// TIA Portal V16 export
// export: Created 2024-05-10T06:46:41.5011859Z, ExportSetting WithDefaults, DisplayName Totally Integrated Automation Portal, DisplayVersion V16, DisplayName TIA Portal Version Control Interface, DisplayVersion V16, DisplayName TIA Portal Openness, DisplayVersion V16, DisplayName STEP 7 Professional, DisplayVersion V16, DisplayName STEP 7 Safety, DisplayVersion V16, DisplayName WinCC Professional, DisplayVersion V16
FUNCTION_BLOCK "K04_报警"   // FB4, LAD
{ S7_Optimized_Access := 'TRUE' }
VERSION : 0.1
// stored: AutoNumber false, IsIECCheckEnabled false, IsRetainMemResEnabled false, MemoryReserve 100, SetENOAutomatically false, UDAEnableTagReadback false
   VAR
      MT_ErrTime : Array[1..3] of IEC_TIMER;   // 故障延迟
   END_VAR
   VAR_TEMP
      "W_All EMO" : Int;   // 急停报警汇总
      "W_All SLC" : Int;   // 光栅报警汇总
      "W_All DSW" : Int;   // 门保报警汇总
      "W_All OtherSafe" : Int;   // 其它安全报警汇总
      "W_All AirALM" : Int;   // 气压报警汇总
      "W_All DrumALM" : Array[1..3] of Int;   // 滚筒故障汇总
      "W_All DrumTiOver" : Array[1..3] of Int;   // 滚筒超时汇总
      "W_All InvALM" : Int;   // 变频器故障汇总
      "W_All InvNoRun" : Int;   // 变频器未运行故障汇总
      "W_All InvOverload" : Int;   // 变频器过载故障汇总
      "W_All InvTiOver" : Int;   // 变频器超时故障汇总
      "W_All ValAdvTiOver" : Array[1..3] of Int;   // 阀出动作超时汇总
      "W_All ValRetTiOver" : Array[1..3] of Int;   // 阀回动作超时汇总
      "W_All ValSensALM" : Array[1..3] of Int;   // 阀到位传感器都ON故障汇总
      "W_All ValSenCroALM" : Array[1..3] of Int;   // 阀到位传感器交叉ON故障汇总
      "W_All AxisALM" : Int;   // 轴报警汇总
      "W_All AxisERR" : Int;   // 轴故障汇总
      "W_All AxisReady" : Int;   // 轴未准备好汇总
      "W_All AxisHomeALM" : Int;   // 轴未回零故障汇总
      "W_All AxisNoRun" : Int;   // 轴未运行汇总
      "W_ALL AxisFLSALM" : Int;   // 轴正极限故障汇总
      "W_All AxisRLSALM" : Int;   // 轴负极限故障汇总
      "W_All RobotALM" : Int;   // 机器人故障汇总
      "W_All CCDALM" : Int;   // 视觉故障汇总
      "W_All CommALM" : Int;   // 通信故障汇总
      "W_All AnalogUpALM" : Int;   // 模拟量上限故障汇总
      "W_All AnalogLowALM" : Int;   // 模拟量下限故障汇总
      "W_All OtherALM" : Int;   // 其它故障汇总
      "W_All SensALM" : Array[1..6] of Int;   // 传感器故障汇总
      "W_All MoveALM" : Array[1..3] of Int;   // 动作异常汇总
      WD_RealTimeALM : Array[1..15] of DInt;   // 故障数据实时
      WD_OldTimeALM : Array[1..10] of DInt;   // 旧的故障
      WD_NewTimeALM : Array[1..10] of DInt;   // 新的故障
      M_SafeType : Bool;   // 安全类别
      M_AirType : Bool;   // 气压类别
      M_DrumType : Bool;   // 滚筒类别
      M_InvType : Bool;   // 变频器类类别
      M_ValType : Bool;   // 电磁阀类别
      M_ServoType : Bool;   // 伺服类别
      M_RoboType : Bool;   // 机器人类别
      M_CCDType : Bool;   // 视觉类别
      M_CommType : Bool;   // 通信类别
      M_AnalogType : Bool;   // 模拟量类别
      M_OtherType : Bool;   // 其它类别
      M_SensType : Bool;   // 传感器类
      M_MoveType : Bool;   // 动作异常类
      "M_All ALM" : Bool;   // 故障汇总
      "M_All NewALM" : Bool;   // 故障汇总新的
      M_BuzzeClose : Bool;   // 故障BZ关闭
      M_Pluse : Array[1..3] of Bool;   // 脉冲
   END_VAR
   VAR_TEMP   // added for the SCL form of the ladder/FBD networks
      _w1 : Bool;
      _w2 : Bool;
      _w3 : Bool;
      _w4 : Bool;
      _w5 : Bool;
      _w6 : Bool;
      _w7 : Bool;
      _w8 : Bool;
      _w9 : Bool;
      _w10 : Bool;
      _w11 : Bool;
      _w12 : Bool;
      _w13 : Bool;
      _w14 : Bool;
      _w15 : Bool;
      _w16 : Bool;
      _w17 : Bool;
      _w18 : Bool;
      _w19 : Bool;
      _w20 : Bool;
      _w21 : Bool;
      _w22 : Bool;
      _w23 : Bool;
      _w24 : Bool;
      _w25 : Bool;
      _w26 : Bool;
      _w27 : Bool;
      _w28 : Bool;
      _w29 : Bool;
      _w30 : Bool;
      _w31 : Bool;
      _w32 : Bool;
      _w33 : Bool;
      _w34 : Bool;
   END_VAR
BEGIN

REGION Network 1: 急停报警16个
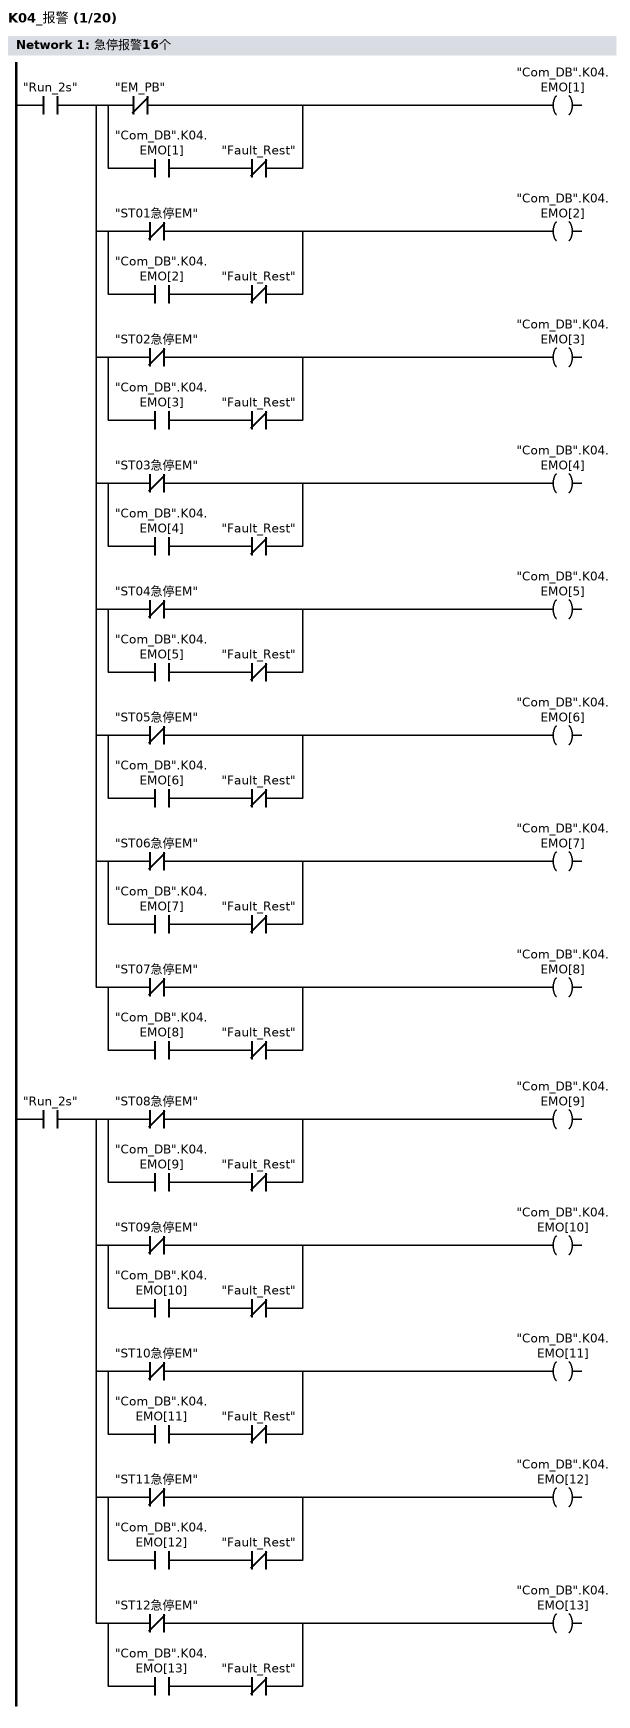
   RUNG wire#powerrail
      Contact( "Run_2s" )
      wire#w1
      I_Contact( "EM_PB" )
      wire#w2
      Coil( "Com_DB".K04.EMO[1] )
   END_RUNG
   RUNG wire#w1
      Contact( "Com_DB".K04.EMO[1] )
      I_Contact( "Fault_Rest" )
   END_RUNG wire#w2
   RUNG wire#w1
      I_Contact( "ST01急停EM" )
      wire#w3
      Coil( "Com_DB".K04.EMO[2] )
   END_RUNG
   RUNG wire#w1
      Contact( "Com_DB".K04.EMO[2] )
      I_Contact( "Fault_Rest" )
   END_RUNG wire#w3
   RUNG wire#w1
      I_Contact( "ST02急停EM" )
      wire#w4
      Coil( "Com_DB".K04.EMO[3] )
   END_RUNG
   RUNG wire#w1
      Contact( "Com_DB".K04.EMO[3] )
      I_Contact( "Fault_Rest" )
   END_RUNG wire#w4
   RUNG wire#w1
      I_Contact( "ST03急停EM" )
      wire#w5
      Coil( "Com_DB".K04.EMO[4] )
   END_RUNG
   RUNG wire#w1
      Contact( "Com_DB".K04.EMO[4] )
      I_Contact( "Fault_Rest" )
   END_RUNG wire#w5
   RUNG wire#w1
      I_Contact( "ST04急停EM" )
      wire#w6
      Coil( "Com_DB".K04.EMO[5] )
   END_RUNG
   RUNG wire#w1
      Contact( "Com_DB".K04.EMO[5] )
      I_Contact( "Fault_Rest" )
   END_RUNG wire#w6
   RUNG wire#w1
      I_Contact( "ST05急停EM" )
      wire#w7
      Coil( "Com_DB".K04.EMO[6] )
   END_RUNG
   RUNG wire#w1
      Contact( "Com_DB".K04.EMO[6] )
      I_Contact( "Fault_Rest" )
   END_RUNG wire#w7
   RUNG wire#w1
      I_Contact( "ST06急停EM" )
      wire#w8
      Coil( "Com_DB".K04.EMO[7] )
   END_RUNG
   RUNG wire#w1
      Contact( "Com_DB".K04.EMO[7] )
      I_Contact( "Fault_Rest" )
   END_RUNG wire#w8
   RUNG wire#w1
      I_Contact( "ST07急停EM" )
      wire#w9
      Coil( "Com_DB".K04.EMO[8] )
   END_RUNG
   RUNG wire#w1
      Contact( "Com_DB".K04.EMO[8] )
      I_Contact( "Fault_Rest" )
   END_RUNG wire#w9
   RUNG wire#powerrail
      Contact( "Run_2s" )
      wire#w10
      I_Contact( "ST08急停EM" )
      wire#w11
      Coil( "Com_DB".K04.EMO[9] )
   END_RUNG
   RUNG wire#w10
      Contact( "Com_DB".K04.EMO[9] )
      I_Contact( "Fault_Rest" )
   END_RUNG wire#w11
   RUNG wire#w10
      I_Contact( "ST09急停EM" )
      wire#w12
      Coil( "Com_DB".K04.EMO[10] )
   END_RUNG
   RUNG wire#w10
      Contact( "Com_DB".K04.EMO[10] )
      I_Contact( "Fault_Rest" )
   END_RUNG wire#w12
   RUNG wire#w10
      I_Contact( "ST10急停EM" )
      wire#w13
      Coil( "Com_DB".K04.EMO[11] )
   END_RUNG
   RUNG wire#w10
      Contact( "Com_DB".K04.EMO[11] )
      I_Contact( "Fault_Rest" )
   END_RUNG wire#w13
   RUNG wire#w10
      I_Contact( "ST11急停EM" )
      wire#w14
      Coil( "Com_DB".K04.EMO[12] )
   END_RUNG
   RUNG wire#w10
      Contact( "Com_DB".K04.EMO[12] )
      I_Contact( "Fault_Rest" )
   END_RUNG wire#w14
   RUNG wire#w10
      I_Contact( "ST12急停EM" )
      wire#w15
      Coil( "Com_DB".K04.EMO[13] )
   END_RUNG
   RUNG wire#w10
      Contact( "Com_DB".K04.EMO[13] )
      I_Contact( "Fault_Rest" )
   END_RUNG wire#w15
   // the same network as SCL:
   "Com_DB".K04.EMO[1] := "Run_2s" AND (NOT "EM_PB" OR ("Com_DB".K04.EMO[1] AND NOT "Fault_Rest"));
   "Com_DB".K04.EMO[2] := "Run_2s" AND (NOT "ST01急停EM" OR ("Com_DB".K04.EMO[2] AND NOT "Fault_Rest"));
   "Com_DB".K04.EMO[3] := "Run_2s" AND (NOT "ST02急停EM" OR ("Com_DB".K04.EMO[3] AND NOT "Fault_Rest"));
   "Com_DB".K04.EMO[4] := "Run_2s" AND (NOT "ST03急停EM" OR ("Com_DB".K04.EMO[4] AND NOT "Fault_Rest"));
   "Com_DB".K04.EMO[5] := "Run_2s" AND (NOT "ST04急停EM" OR ("Com_DB".K04.EMO[5] AND NOT "Fault_Rest"));
   "Com_DB".K04.EMO[6] := "Run_2s" AND (NOT "ST05急停EM" OR ("Com_DB".K04.EMO[6] AND NOT "Fault_Rest"));
   "Com_DB".K04.EMO[7] := "Run_2s" AND (NOT "ST06急停EM" OR ("Com_DB".K04.EMO[7] AND NOT "Fault_Rest"));
   "Com_DB".K04.EMO[8] := "Run_2s" AND (NOT "ST07急停EM" OR ("Com_DB".K04.EMO[8] AND NOT "Fault_Rest"));
   "Com_DB".K04.EMO[9] := "Run_2s" AND (NOT "ST08急停EM" OR ("Com_DB".K04.EMO[9] AND NOT "Fault_Rest"));
   "Com_DB".K04.EMO[10] := "Run_2s" AND (NOT "ST09急停EM" OR ("Com_DB".K04.EMO[10] AND NOT "Fault_Rest"));
   "Com_DB".K04.EMO[11] := "Run_2s" AND (NOT "ST10急停EM" OR ("Com_DB".K04.EMO[11] AND NOT "Fault_Rest"));
   "Com_DB".K04.EMO[12] := "Run_2s" AND (NOT "ST11急停EM" OR ("Com_DB".K04.EMO[12] AND NOT "Fault_Rest"));
   "Com_DB".K04.EMO[13] := "Run_2s" AND (NOT "ST12急停EM" OR ("Com_DB".K04.EMO[13] AND NOT "Fault_Rest"));
END_REGION

REGION Network 2: 光栅报警16个
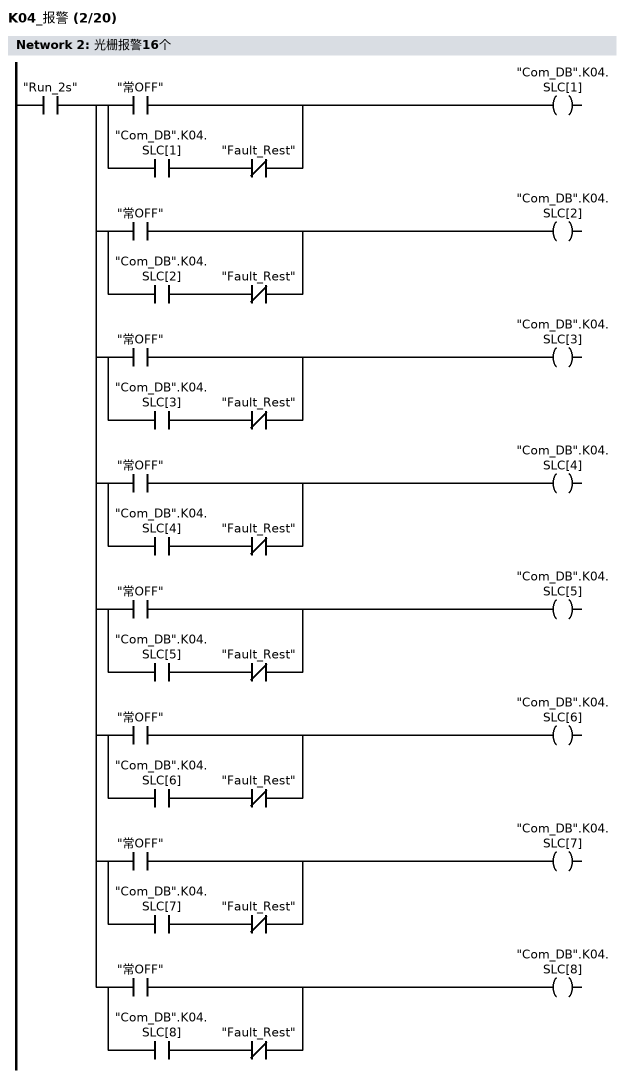
   RUNG wire#powerrail
      Contact( "Run_2s" )
      wire#w1
      Contact( "常OFF" )
      wire#w2
      Coil( "Com_DB".K04.SLC[1] )
   END_RUNG
   RUNG wire#w1
      Contact( "Com_DB".K04.SLC[1] )
      I_Contact( "Fault_Rest" )
   END_RUNG wire#w2
   RUNG wire#w1
      Contact( "常OFF" )
      wire#w3
      Coil( "Com_DB".K04.SLC[2] )
   END_RUNG
   RUNG wire#w1
      Contact( "Com_DB".K04.SLC[2] )
      I_Contact( "Fault_Rest" )
   END_RUNG wire#w3
   RUNG wire#w1
      Contact( "常OFF" )
      wire#w4
      Coil( "Com_DB".K04.SLC[3] )
   END_RUNG
   RUNG wire#w1
      Contact( "Com_DB".K04.SLC[3] )
      I_Contact( "Fault_Rest" )
   END_RUNG wire#w4
   RUNG wire#w1
      Contact( "常OFF" )
      wire#w5
      Coil( "Com_DB".K04.SLC[4] )
   END_RUNG
   RUNG wire#w1
      Contact( "Com_DB".K04.SLC[4] )
      I_Contact( "Fault_Rest" )
   END_RUNG wire#w5
   RUNG wire#w1
      Contact( "常OFF" )
      wire#w6
      Coil( "Com_DB".K04.SLC[5] )
   END_RUNG
   RUNG wire#w1
      Contact( "Com_DB".K04.SLC[5] )
      I_Contact( "Fault_Rest" )
   END_RUNG wire#w6
   RUNG wire#w1
      Contact( "常OFF" )
      wire#w7
      Coil( "Com_DB".K04.SLC[6] )
   END_RUNG
   RUNG wire#w1
      Contact( "Com_DB".K04.SLC[6] )
      I_Contact( "Fault_Rest" )
   END_RUNG wire#w7
   RUNG wire#w1
      Contact( "常OFF" )
      wire#w8
      Coil( "Com_DB".K04.SLC[7] )
   END_RUNG
   RUNG wire#w1
      Contact( "Com_DB".K04.SLC[7] )
      I_Contact( "Fault_Rest" )
   END_RUNG wire#w8
   RUNG wire#w1
      Contact( "常OFF" )
      wire#w9
      Coil( "Com_DB".K04.SLC[8] )
   END_RUNG
   RUNG wire#w1
      Contact( "Com_DB".K04.SLC[8] )
      I_Contact( "Fault_Rest" )
   END_RUNG wire#w9
   // the same network as SCL:
   "Com_DB".K04.SLC[1] := "Run_2s" AND ("常OFF" OR ("Com_DB".K04.SLC[1] AND NOT "Fault_Rest"));
   "Com_DB".K04.SLC[2] := "Run_2s" AND ("常OFF" OR ("Com_DB".K04.SLC[2] AND NOT "Fault_Rest"));
   "Com_DB".K04.SLC[3] := "Run_2s" AND ("常OFF" OR ("Com_DB".K04.SLC[3] AND NOT "Fault_Rest"));
   "Com_DB".K04.SLC[4] := "Run_2s" AND ("常OFF" OR ("Com_DB".K04.SLC[4] AND NOT "Fault_Rest"));
   "Com_DB".K04.SLC[5] := "Run_2s" AND ("常OFF" OR ("Com_DB".K04.SLC[5] AND NOT "Fault_Rest"));
   "Com_DB".K04.SLC[6] := "Run_2s" AND ("常OFF" OR ("Com_DB".K04.SLC[6] AND NOT "Fault_Rest"));
   "Com_DB".K04.SLC[7] := "Run_2s" AND ("常OFF" OR ("Com_DB".K04.SLC[7] AND NOT "Fault_Rest"));
   "Com_DB".K04.SLC[8] := "Run_2s" AND ("常OFF" OR ("Com_DB".K04.SLC[8] AND NOT "Fault_Rest"));
END_REGION

REGION Network 3: 门开关报警16个
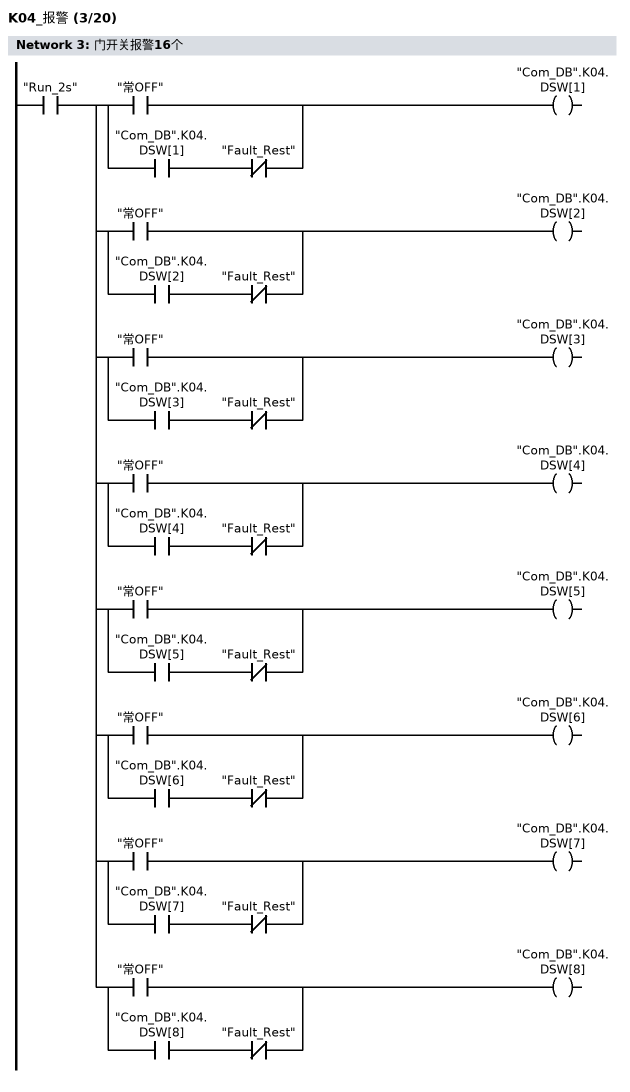
   RUNG wire#powerrail
      Contact( "Run_2s" )
      wire#w1
      Contact( "常OFF" )
      wire#w2
      Coil( "Com_DB".K04.DSW[1] )
   END_RUNG
   RUNG wire#w1
      Contact( "Com_DB".K04.DSW[1] )
      I_Contact( "Fault_Rest" )
   END_RUNG wire#w2
   RUNG wire#w1
      Contact( "常OFF" )
      wire#w3
      Coil( "Com_DB".K04.DSW[2] )
   END_RUNG
   RUNG wire#w1
      Contact( "Com_DB".K04.DSW[2] )
      I_Contact( "Fault_Rest" )
   END_RUNG wire#w3
   RUNG wire#w1
      Contact( "常OFF" )
      wire#w4
      Coil( "Com_DB".K04.DSW[3] )
   END_RUNG
   RUNG wire#w1
      Contact( "Com_DB".K04.DSW[3] )
      I_Contact( "Fault_Rest" )
   END_RUNG wire#w4
   RUNG wire#w1
      Contact( "常OFF" )
      wire#w5
      Coil( "Com_DB".K04.DSW[4] )
   END_RUNG
   RUNG wire#w1
      Contact( "Com_DB".K04.DSW[4] )
      I_Contact( "Fault_Rest" )
   END_RUNG wire#w5
   RUNG wire#w1
      Contact( "常OFF" )
      wire#w6
      Coil( "Com_DB".K04.DSW[5] )
   END_RUNG
   RUNG wire#w1
      Contact( "Com_DB".K04.DSW[5] )
      I_Contact( "Fault_Rest" )
   END_RUNG wire#w6
   RUNG wire#w1
      Contact( "常OFF" )
      wire#w7
      Coil( "Com_DB".K04.DSW[6] )
   END_RUNG
   RUNG wire#w1
      Contact( "Com_DB".K04.DSW[6] )
      I_Contact( "Fault_Rest" )
   END_RUNG wire#w7
   RUNG wire#w1
      Contact( "常OFF" )
      wire#w8
      Coil( "Com_DB".K04.DSW[7] )
   END_RUNG
   RUNG wire#w1
      Contact( "Com_DB".K04.DSW[7] )
      I_Contact( "Fault_Rest" )
   END_RUNG wire#w8
   RUNG wire#w1
      Contact( "常OFF" )
      wire#w9
      Coil( "Com_DB".K04.DSW[8] )
   END_RUNG
   RUNG wire#w1
      Contact( "Com_DB".K04.DSW[8] )
      I_Contact( "Fault_Rest" )
   END_RUNG wire#w9
   // the same network as SCL:
   "Com_DB".K04.DSW[1] := "Run_2s" AND ("常OFF" OR ("Com_DB".K04.DSW[1] AND NOT "Fault_Rest"));
   "Com_DB".K04.DSW[2] := "Run_2s" AND ("常OFF" OR ("Com_DB".K04.DSW[2] AND NOT "Fault_Rest"));
   "Com_DB".K04.DSW[3] := "Run_2s" AND ("常OFF" OR ("Com_DB".K04.DSW[3] AND NOT "Fault_Rest"));
   "Com_DB".K04.DSW[4] := "Run_2s" AND ("常OFF" OR ("Com_DB".K04.DSW[4] AND NOT "Fault_Rest"));
   "Com_DB".K04.DSW[5] := "Run_2s" AND ("常OFF" OR ("Com_DB".K04.DSW[5] AND NOT "Fault_Rest"));
   "Com_DB".K04.DSW[6] := "Run_2s" AND ("常OFF" OR ("Com_DB".K04.DSW[6] AND NOT "Fault_Rest"));
   "Com_DB".K04.DSW[7] := "Run_2s" AND ("常OFF" OR ("Com_DB".K04.DSW[7] AND NOT "Fault_Rest"));
   "Com_DB".K04.DSW[8] := "Run_2s" AND ("常OFF" OR ("Com_DB".K04.DSW[8] AND NOT "Fault_Rest"));
END_REGION

REGION Network 4: 其它安全报警16个Other types of security
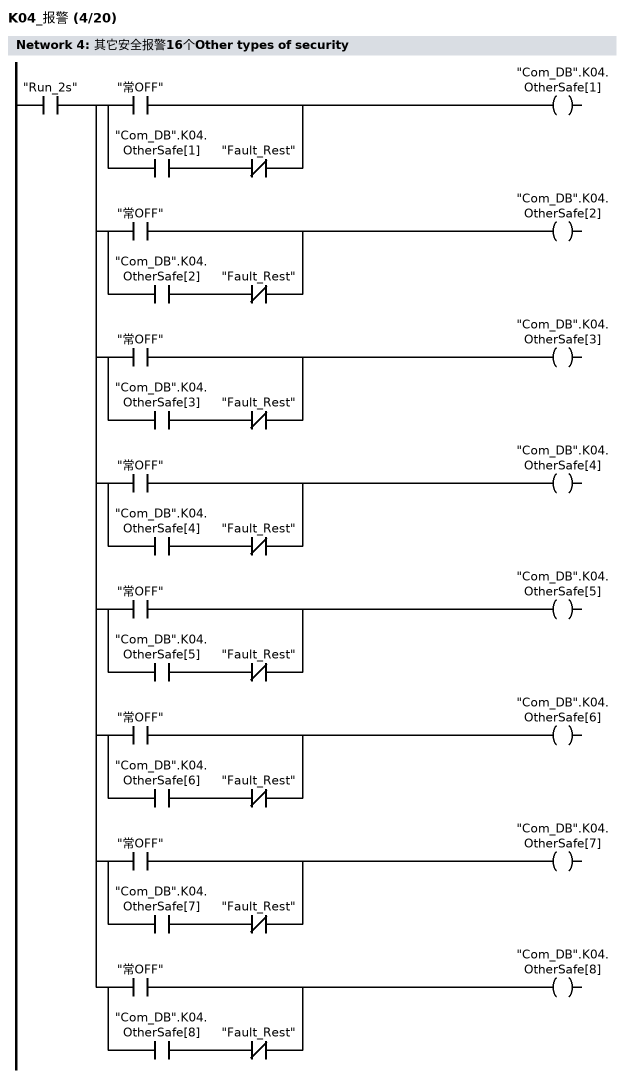
   RUNG wire#powerrail
      Contact( "Run_2s" )
      wire#w1
      Contact( "常OFF" )
      wire#w2
      Coil( "Com_DB".K04.OtherSafe[1] )
   END_RUNG
   RUNG wire#w1
      Contact( "Com_DB".K04.OtherSafe[1] )
      I_Contact( "Fault_Rest" )
   END_RUNG wire#w2
   RUNG wire#w1
      Contact( "常OFF" )
      wire#w3
      Coil( "Com_DB".K04.OtherSafe[2] )
   END_RUNG
   RUNG wire#w1
      Contact( "Com_DB".K04.OtherSafe[2] )
      I_Contact( "Fault_Rest" )
   END_RUNG wire#w3
   RUNG wire#w1
      Contact( "常OFF" )
      wire#w4
      Coil( "Com_DB".K04.OtherSafe[3] )
   END_RUNG
   RUNG wire#w1
      Contact( "Com_DB".K04.OtherSafe[3] )
      I_Contact( "Fault_Rest" )
   END_RUNG wire#w4
   RUNG wire#w1
      Contact( "常OFF" )
      wire#w5
      Coil( "Com_DB".K04.OtherSafe[4] )
   END_RUNG
   RUNG wire#w1
      Contact( "Com_DB".K04.OtherSafe[4] )
      I_Contact( "Fault_Rest" )
   END_RUNG wire#w5
   RUNG wire#w1
      Contact( "常OFF" )
      wire#w6
      Coil( "Com_DB".K04.OtherSafe[5] )
   END_RUNG
   RUNG wire#w1
      Contact( "Com_DB".K04.OtherSafe[5] )
      I_Contact( "Fault_Rest" )
   END_RUNG wire#w6
   RUNG wire#w1
      Contact( "常OFF" )
      wire#w7
      Coil( "Com_DB".K04.OtherSafe[6] )
   END_RUNG
   RUNG wire#w1
      Contact( "Com_DB".K04.OtherSafe[6] )
      I_Contact( "Fault_Rest" )
   END_RUNG wire#w7
   RUNG wire#w1
      Contact( "常OFF" )
      wire#w8
      Coil( "Com_DB".K04.OtherSafe[7] )
   END_RUNG
   RUNG wire#w1
      Contact( "Com_DB".K04.OtherSafe[7] )
      I_Contact( "Fault_Rest" )
   END_RUNG wire#w8
   RUNG wire#w1
      Contact( "常OFF" )
      wire#w9
      Coil( "Com_DB".K04.OtherSafe[8] )
   END_RUNG
   RUNG wire#w1
      Contact( "Com_DB".K04.OtherSafe[8] )
      I_Contact( "Fault_Rest" )
   END_RUNG wire#w9
   // the same network as SCL:
   "Com_DB".K04.OtherSafe[1] := "Run_2s" AND ("常OFF" OR ("Com_DB".K04.OtherSafe[1] AND NOT "Fault_Rest"));
   "Com_DB".K04.OtherSafe[2] := "Run_2s" AND ("常OFF" OR ("Com_DB".K04.OtherSafe[2] AND NOT "Fault_Rest"));
   "Com_DB".K04.OtherSafe[3] := "Run_2s" AND ("常OFF" OR ("Com_DB".K04.OtherSafe[3] AND NOT "Fault_Rest"));
   "Com_DB".K04.OtherSafe[4] := "Run_2s" AND ("常OFF" OR ("Com_DB".K04.OtherSafe[4] AND NOT "Fault_Rest"));
   "Com_DB".K04.OtherSafe[5] := "Run_2s" AND ("常OFF" OR ("Com_DB".K04.OtherSafe[5] AND NOT "Fault_Rest"));
   "Com_DB".K04.OtherSafe[6] := "Run_2s" AND ("常OFF" OR ("Com_DB".K04.OtherSafe[6] AND NOT "Fault_Rest"));
   "Com_DB".K04.OtherSafe[7] := "Run_2s" AND ("常OFF" OR ("Com_DB".K04.OtherSafe[7] AND NOT "Fault_Rest"));
   "Com_DB".K04.OtherSafe[8] := "Run_2s" AND ("常OFF" OR ("Com_DB".K04.OtherSafe[8] AND NOT "Fault_Rest"));
END_REGION

REGION Network 5: 气压低报警16个
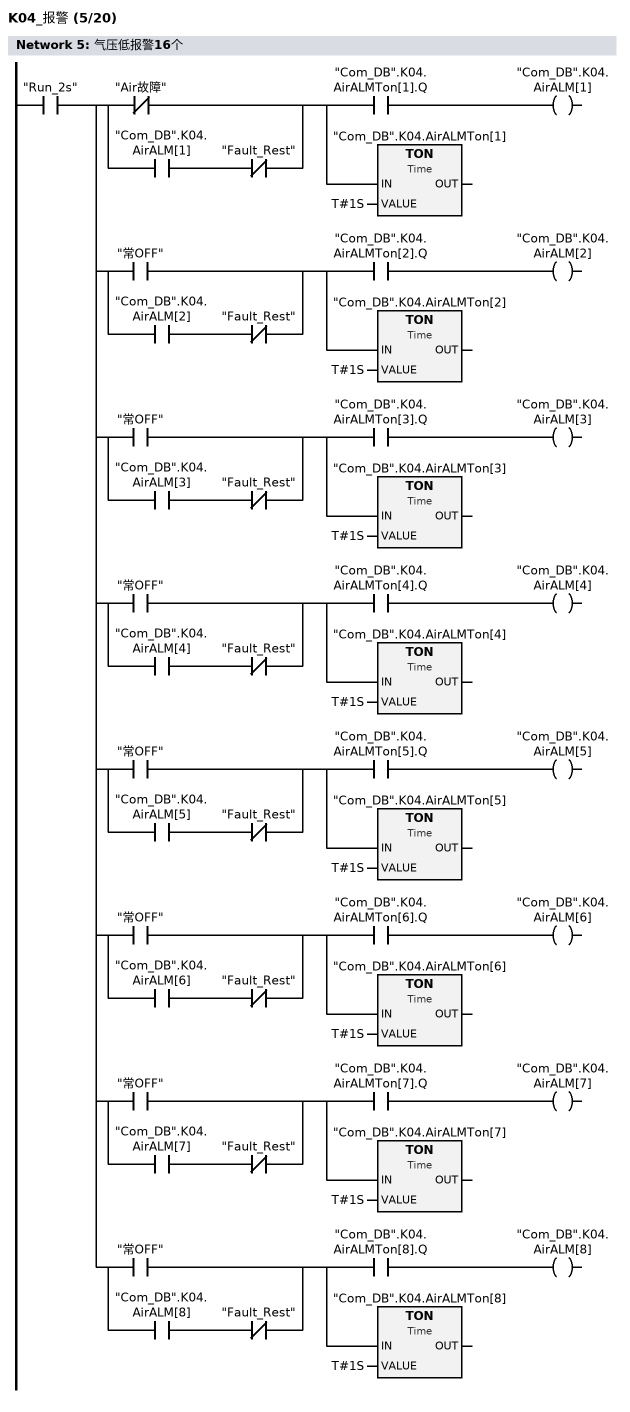
   #_w1 := "Run_2s" AND (NOT "Air故障" OR ("Com_DB".K04.AirALM[1] AND NOT "Fault_Rest"));
   "Com_DB".K04.AirALM[1] := #_w1 AND "Com_DB".K04.AirALMTon[1].Q;
   "Com_DB".K04.AirALMTon[1].TON(IN := #_w1, PT := T#1S);   // TON coil
   #_w2 := "Run_2s" AND ("常OFF" OR ("Com_DB".K04.AirALM[2] AND NOT "Fault_Rest"));
   "Com_DB".K04.AirALM[2] := #_w2 AND "Com_DB".K04.AirALMTon[2].Q;
   "Com_DB".K04.AirALMTon[2].TON(IN := #_w2, PT := T#1S);   // TON coil
   #_w3 := "Run_2s" AND ("常OFF" OR ("Com_DB".K04.AirALM[3] AND NOT "Fault_Rest"));
   "Com_DB".K04.AirALM[3] := #_w3 AND "Com_DB".K04.AirALMTon[3].Q;
   "Com_DB".K04.AirALMTon[3].TON(IN := #_w3, PT := T#1S);   // TON coil
   #_w4 := "Run_2s" AND ("常OFF" OR ("Com_DB".K04.AirALM[4] AND NOT "Fault_Rest"));
   "Com_DB".K04.AirALM[4] := #_w4 AND "Com_DB".K04.AirALMTon[4].Q;
   "Com_DB".K04.AirALMTon[4].TON(IN := #_w4, PT := T#1S);   // TON coil
   #_w5 := "Run_2s" AND ("常OFF" OR ("Com_DB".K04.AirALM[5] AND NOT "Fault_Rest"));
   "Com_DB".K04.AirALM[5] := #_w5 AND "Com_DB".K04.AirALMTon[5].Q;
   "Com_DB".K04.AirALMTon[5].TON(IN := #_w5, PT := T#1S);   // TON coil
   #_w6 := "Run_2s" AND ("常OFF" OR ("Com_DB".K04.AirALM[6] AND NOT "Fault_Rest"));
   "Com_DB".K04.AirALM[6] := #_w6 AND "Com_DB".K04.AirALMTon[6].Q;
   "Com_DB".K04.AirALMTon[6].TON(IN := #_w6, PT := T#1S);   // TON coil
   #_w7 := "Run_2s" AND ("常OFF" OR ("Com_DB".K04.AirALM[7] AND NOT "Fault_Rest"));
   "Com_DB".K04.AirALM[7] := #_w7 AND "Com_DB".K04.AirALMTon[7].Q;
   "Com_DB".K04.AirALMTon[7].TON(IN := #_w7, PT := T#1S);   // TON coil
   #_w8 := "Run_2s" AND ("常OFF" OR ("Com_DB".K04.AirALM[8] AND NOT "Fault_Rest"));
   "Com_DB".K04.AirALM[8] := #_w8 AND "Com_DB".K04.AirALMTon[8].Q;
   "Com_DB".K04.AirALMTon[8].TON(IN := #_w8, PT := T#1S);   // TON coil
END_REGION

REGION Network 6: 滚筒故障48个
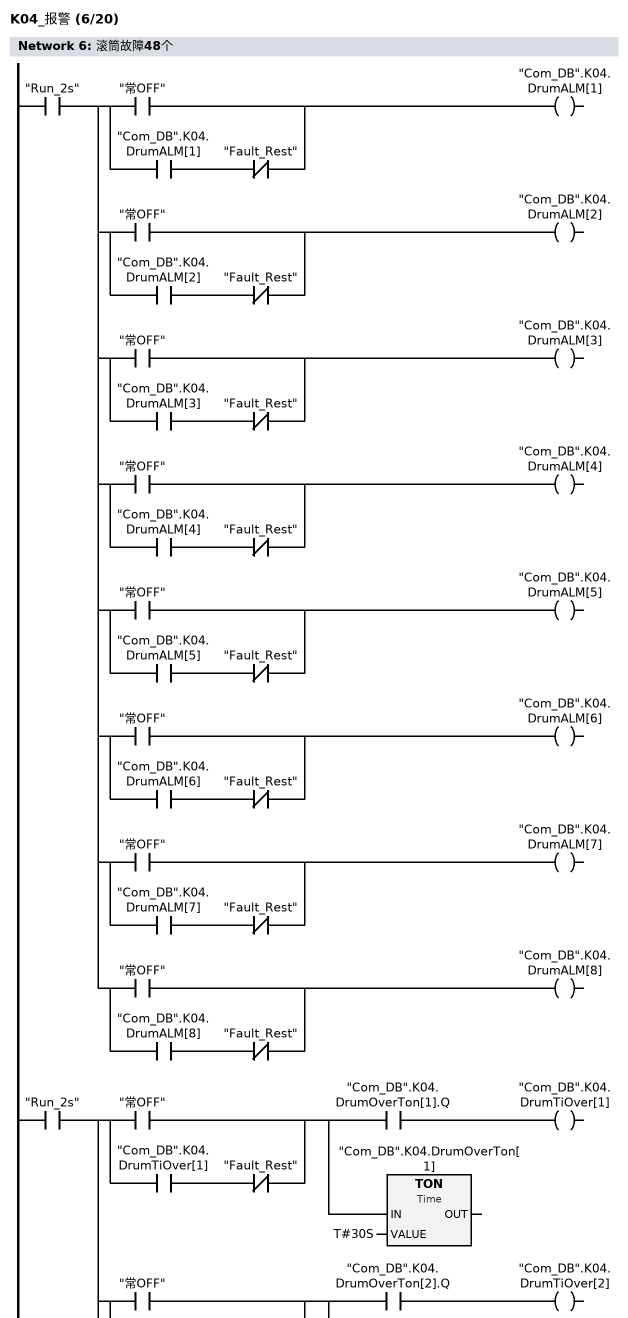
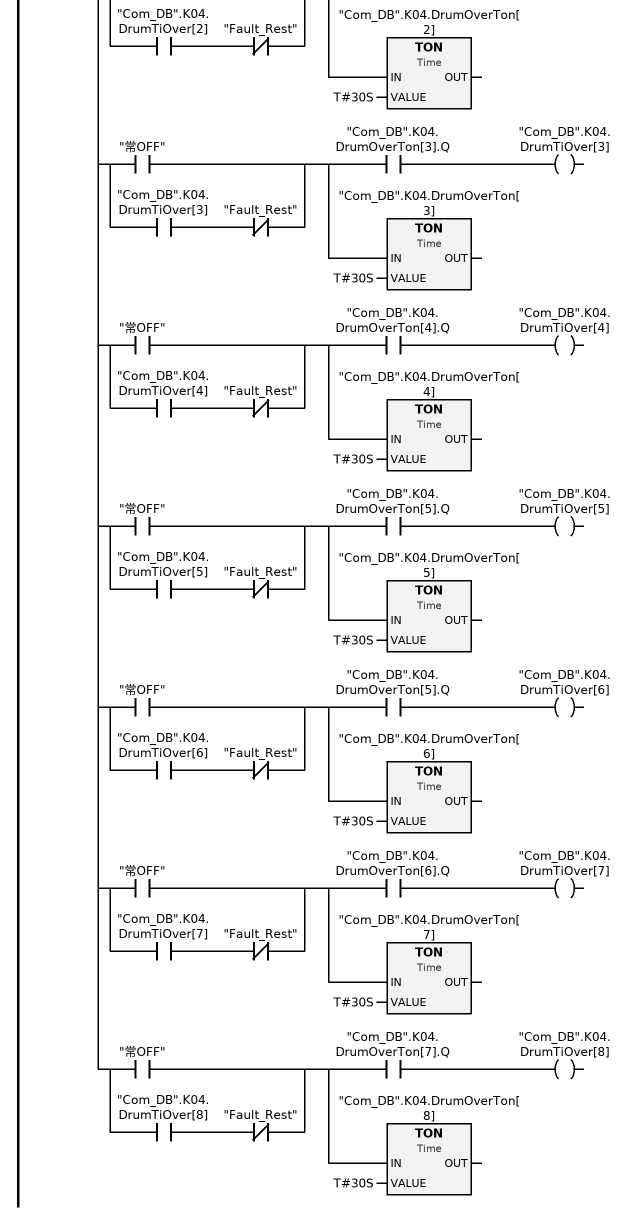
   "Com_DB".K04.DrumALM[1] := "Run_2s" AND ("常OFF" OR ("Com_DB".K04.DrumALM[1] AND NOT "Fault_Rest"));
   "Com_DB".K04.DrumALM[2] := "Run_2s" AND ("常OFF" OR ("Com_DB".K04.DrumALM[2] AND NOT "Fault_Rest"));
   "Com_DB".K04.DrumALM[3] := "Run_2s" AND ("常OFF" OR ("Com_DB".K04.DrumALM[3] AND NOT "Fault_Rest"));
   "Com_DB".K04.DrumALM[4] := "Run_2s" AND ("常OFF" OR ("Com_DB".K04.DrumALM[4] AND NOT "Fault_Rest"));
   "Com_DB".K04.DrumALM[5] := "Run_2s" AND ("常OFF" OR ("Com_DB".K04.DrumALM[5] AND NOT "Fault_Rest"));
   "Com_DB".K04.DrumALM[6] := "Run_2s" AND ("常OFF" OR ("Com_DB".K04.DrumALM[6] AND NOT "Fault_Rest"));
   "Com_DB".K04.DrumALM[7] := "Run_2s" AND ("常OFF" OR ("Com_DB".K04.DrumALM[7] AND NOT "Fault_Rest"));
   "Com_DB".K04.DrumALM[8] := "Run_2s" AND ("常OFF" OR ("Com_DB".K04.DrumALM[8] AND NOT "Fault_Rest"));
   #_w1 := "Run_2s" AND ("常OFF" OR ("Com_DB".K04.DrumTiOver[1] AND NOT "Fault_Rest"));
   "Com_DB".K04.DrumTiOver[1] := #_w1 AND "Com_DB".K04.DrumOverTon[1].Q;
   "Com_DB".K04.DrumOverTon[1].TON(IN := #_w1, PT := T#30S);   // TON coil
   #_w2 := "Run_2s" AND ("常OFF" OR ("Com_DB".K04.DrumTiOver[2] AND NOT "Fault_Rest"));
   "Com_DB".K04.DrumTiOver[2] := #_w2 AND "Com_DB".K04.DrumOverTon[2].Q;
   "Com_DB".K04.DrumOverTon[2].TON(IN := #_w2, PT := T#30S);   // TON coil
   #_w3 := "Run_2s" AND ("常OFF" OR ("Com_DB".K04.DrumTiOver[3] AND NOT "Fault_Rest"));
   "Com_DB".K04.DrumTiOver[3] := #_w3 AND "Com_DB".K04.DrumOverTon[3].Q;
   "Com_DB".K04.DrumOverTon[3].TON(IN := #_w3, PT := T#30S);   // TON coil
   #_w4 := "Run_2s" AND ("常OFF" OR ("Com_DB".K04.DrumTiOver[4] AND NOT "Fault_Rest"));
   "Com_DB".K04.DrumTiOver[4] := #_w4 AND "Com_DB".K04.DrumOverTon[4].Q;
   "Com_DB".K04.DrumOverTon[4].TON(IN := #_w4, PT := T#30S);   // TON coil
   #_w5 := "Run_2s" AND ("常OFF" OR ("Com_DB".K04.DrumTiOver[5] AND NOT "Fault_Rest"));
   "Com_DB".K04.DrumTiOver[5] := #_w5 AND "Com_DB".K04.DrumOverTon[5].Q;
   "Com_DB".K04.DrumOverTon[5].TON(IN := #_w5, PT := T#30S);   // TON coil
   #_w6 := "Run_2s" AND ("常OFF" OR ("Com_DB".K04.DrumTiOver[6] AND NOT "Fault_Rest"));
   "Com_DB".K04.DrumTiOver[6] := #_w6 AND "Com_DB".K04.DrumOverTon[5].Q;
   "Com_DB".K04.DrumOverTon[6].TON(IN := #_w6, PT := T#30S);   // TON coil
   #_w7 := "Run_2s" AND ("常OFF" OR ("Com_DB".K04.DrumTiOver[7] AND NOT "Fault_Rest"));
   "Com_DB".K04.DrumTiOver[7] := #_w7 AND "Com_DB".K04.DrumOverTon[6].Q;
   "Com_DB".K04.DrumOverTon[7].TON(IN := #_w7, PT := T#30S);   // TON coil
   #_w8 := "Run_2s" AND ("常OFF" OR ("Com_DB".K04.DrumTiOver[8] AND NOT "Fault_Rest"));
   "Com_DB".K04.DrumTiOver[8] := #_w8 AND "Com_DB".K04.DrumOverTon[7].Q;
   "Com_DB".K04.DrumOverTon[8].TON(IN := #_w8, PT := T#30S);   // TON coil
END_REGION

REGION Network 7: 变频器 异常/未运/超时/过载 16个
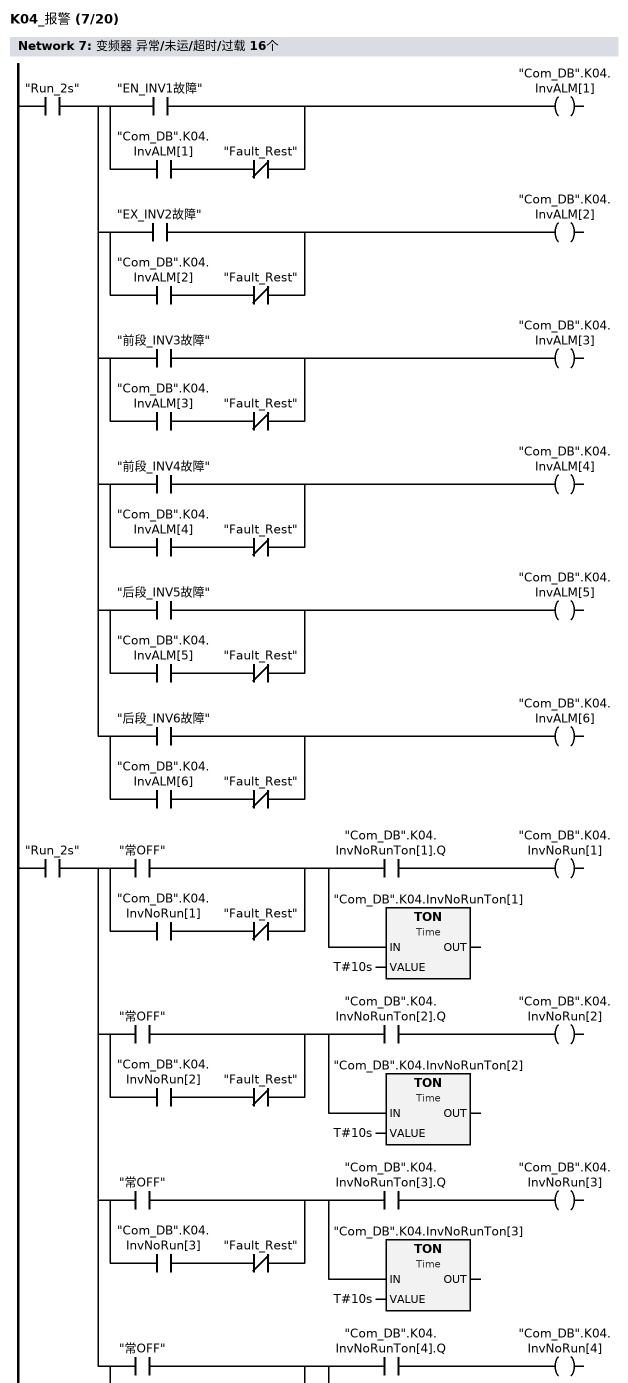
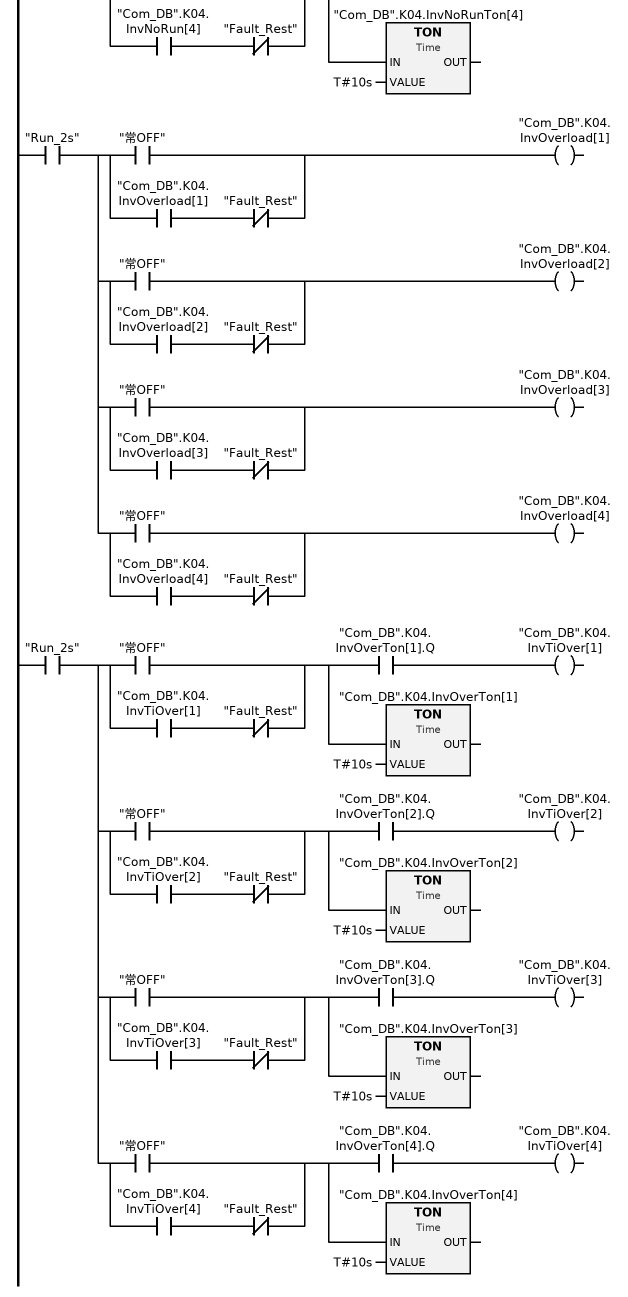
   "Com_DB".K04.InvALM[1] := "Run_2s" AND ("EN_INV1故障" OR ("Com_DB".K04.InvALM[1] AND NOT "Fault_Rest"));
   "Com_DB".K04.InvALM[2] := "Run_2s" AND ("EX_INV2故障" OR ("Com_DB".K04.InvALM[2] AND NOT "Fault_Rest"));
   "Com_DB".K04.InvALM[3] := "Run_2s" AND ("前段_INV3故障" OR ("Com_DB".K04.InvALM[3] AND NOT "Fault_Rest"));
   "Com_DB".K04.InvALM[4] := "Run_2s" AND ("前段_INV4故障" OR ("Com_DB".K04.InvALM[4] AND NOT "Fault_Rest"));
   "Com_DB".K04.InvALM[5] := "Run_2s" AND ("后段_INV5故障" OR ("Com_DB".K04.InvALM[5] AND NOT "Fault_Rest"));
   "Com_DB".K04.InvALM[6] := "Run_2s" AND ("后段_INV6故障" OR ("Com_DB".K04.InvALM[6] AND NOT "Fault_Rest"));
   #_w1 := "Run_2s" AND ("常OFF" OR ("Com_DB".K04.InvNoRun[1] AND NOT "Fault_Rest"));
   "Com_DB".K04.InvNoRun[1] := #_w1 AND "Com_DB".K04.InvNoRunTon[1].Q;
   "Com_DB".K04.InvNoRunTon[1].TON(IN := #_w1, PT := T#10s);   // TON coil
   #_w2 := "Run_2s" AND ("常OFF" OR ("Com_DB".K04.InvNoRun[2] AND NOT "Fault_Rest"));
   "Com_DB".K04.InvNoRun[2] := #_w2 AND "Com_DB".K04.InvNoRunTon[2].Q;
   "Com_DB".K04.InvNoRunTon[2].TON(IN := #_w2, PT := T#10s);   // TON coil
   #_w3 := "Run_2s" AND ("常OFF" OR ("Com_DB".K04.InvNoRun[3] AND NOT "Fault_Rest"));
   "Com_DB".K04.InvNoRun[3] := #_w3 AND "Com_DB".K04.InvNoRunTon[3].Q;
   "Com_DB".K04.InvNoRunTon[3].TON(IN := #_w3, PT := T#10s);   // TON coil
   #_w4 := "Run_2s" AND ("常OFF" OR ("Com_DB".K04.InvNoRun[4] AND NOT "Fault_Rest"));
   "Com_DB".K04.InvNoRun[4] := #_w4 AND "Com_DB".K04.InvNoRunTon[4].Q;
   "Com_DB".K04.InvNoRunTon[4].TON(IN := #_w4, PT := T#10s);   // TON coil
   "Com_DB".K04.InvOverload[1] := "Run_2s" AND ("常OFF" OR ("Com_DB".K04.InvOverload[1] AND NOT "Fault_Rest"));
   "Com_DB".K04.InvOverload[2] := "Run_2s" AND ("常OFF" OR ("Com_DB".K04.InvOverload[2] AND NOT "Fault_Rest"));
   "Com_DB".K04.InvOverload[3] := "Run_2s" AND ("常OFF" OR ("Com_DB".K04.InvOverload[3] AND NOT "Fault_Rest"));
   "Com_DB".K04.InvOverload[4] := "Run_2s" AND ("常OFF" OR ("Com_DB".K04.InvOverload[4] AND NOT "Fault_Rest"));
   #_w5 := "Run_2s" AND ("常OFF" OR ("Com_DB".K04.InvTiOver[1] AND NOT "Fault_Rest"));
   "Com_DB".K04.InvTiOver[1] := #_w5 AND "Com_DB".K04.InvOverTon[1].Q;
   "Com_DB".K04.InvOverTon[1].TON(IN := #_w5, PT := T#10s);   // TON coil
   #_w6 := "Run_2s" AND ("常OFF" OR ("Com_DB".K04.InvTiOver[2] AND NOT "Fault_Rest"));
   "Com_DB".K04.InvTiOver[2] := #_w6 AND "Com_DB".K04.InvOverTon[2].Q;
   "Com_DB".K04.InvOverTon[2].TON(IN := #_w6, PT := T#10s);   // TON coil
   #_w7 := "Run_2s" AND ("常OFF" OR ("Com_DB".K04.InvTiOver[3] AND NOT "Fault_Rest"));
   "Com_DB".K04.InvTiOver[3] := #_w7 AND "Com_DB".K04.InvOverTon[3].Q;
   "Com_DB".K04.InvOverTon[3].TON(IN := #_w7, PT := T#10s);   // TON coil
   #_w8 := "Run_2s" AND ("常OFF" OR ("Com_DB".K04.InvTiOver[4] AND NOT "Fault_Rest"));
   "Com_DB".K04.InvTiOver[4] := #_w8 AND "Com_DB".K04.InvOverTon[4].Q;
   "Com_DB".K04.InvOverTon[4].TON(IN := #_w8, PT := T#10s);   // TON coil
END_REGION

REGION Network 8: 气缸故障48个
   // 气缸故障FB库已经有输出故障，请在FB关联，这里不需写
END_REGION

REGION Network 9: 伺服故障16个伺服
   // 轴警告、轴错误FB库以及有输出，这里不需要写
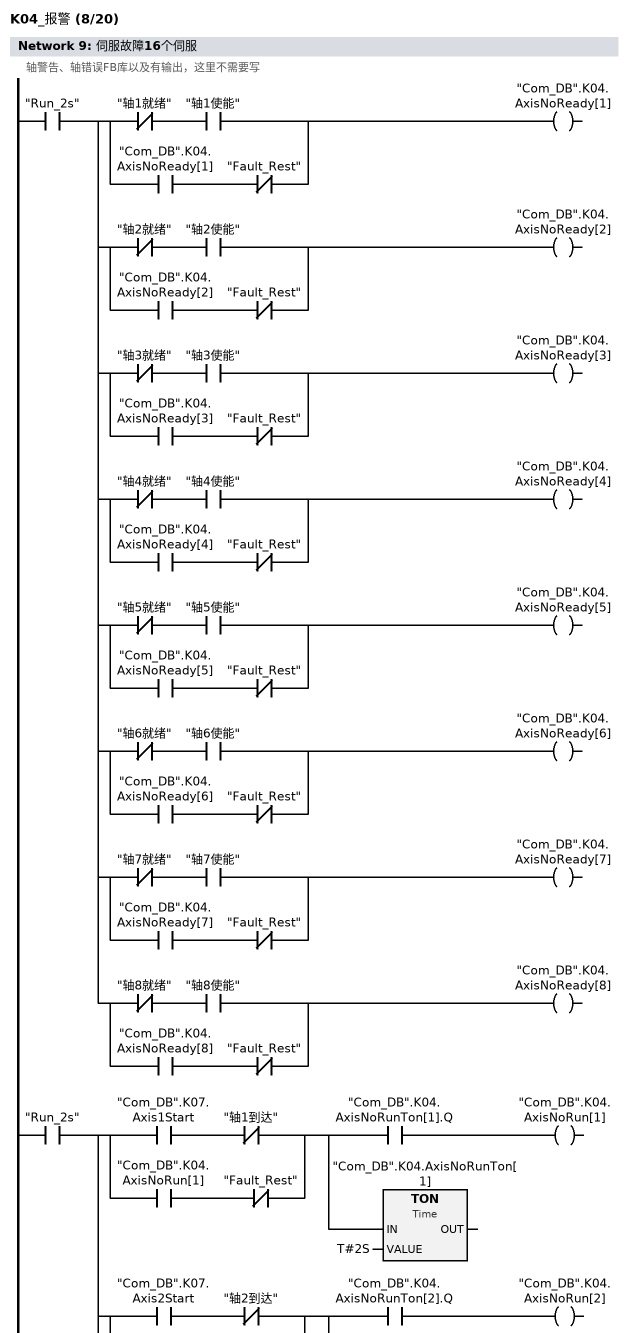
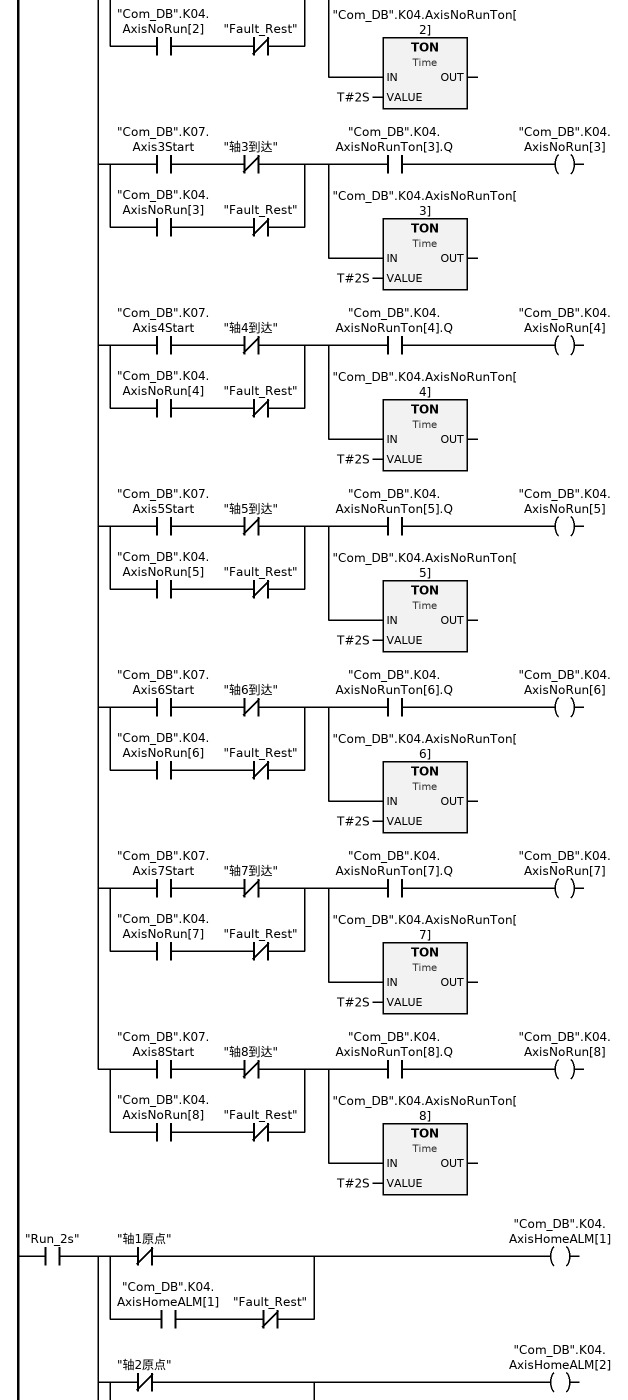
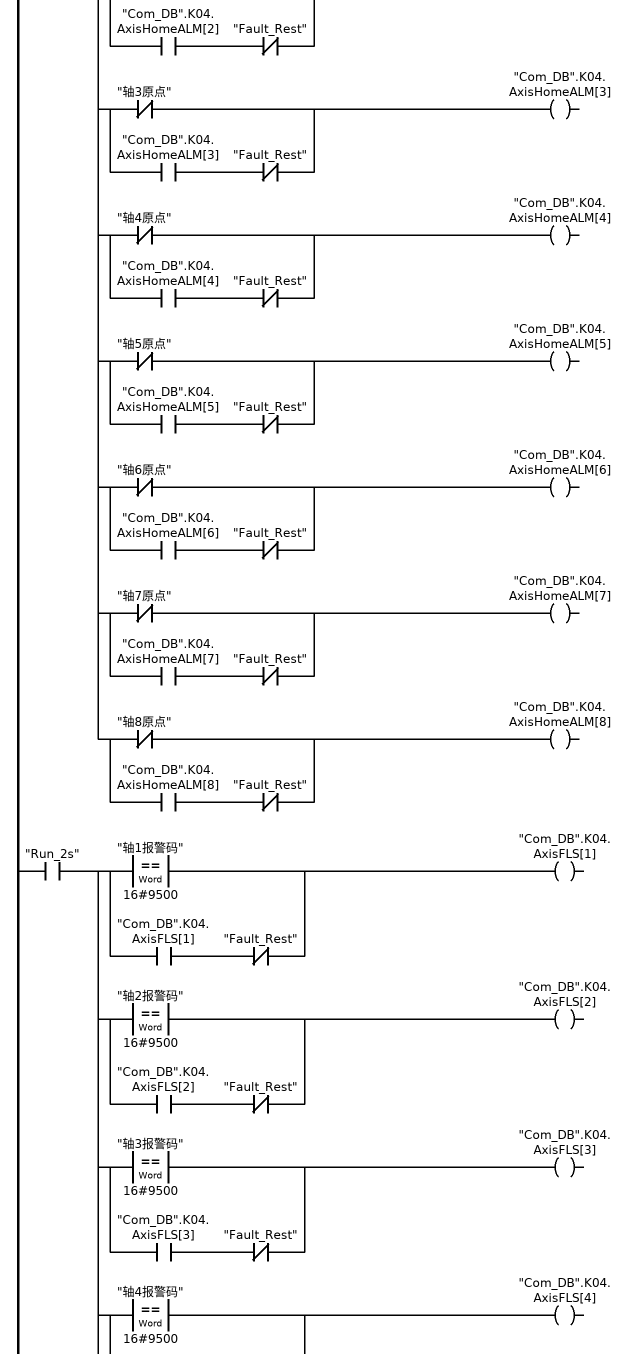
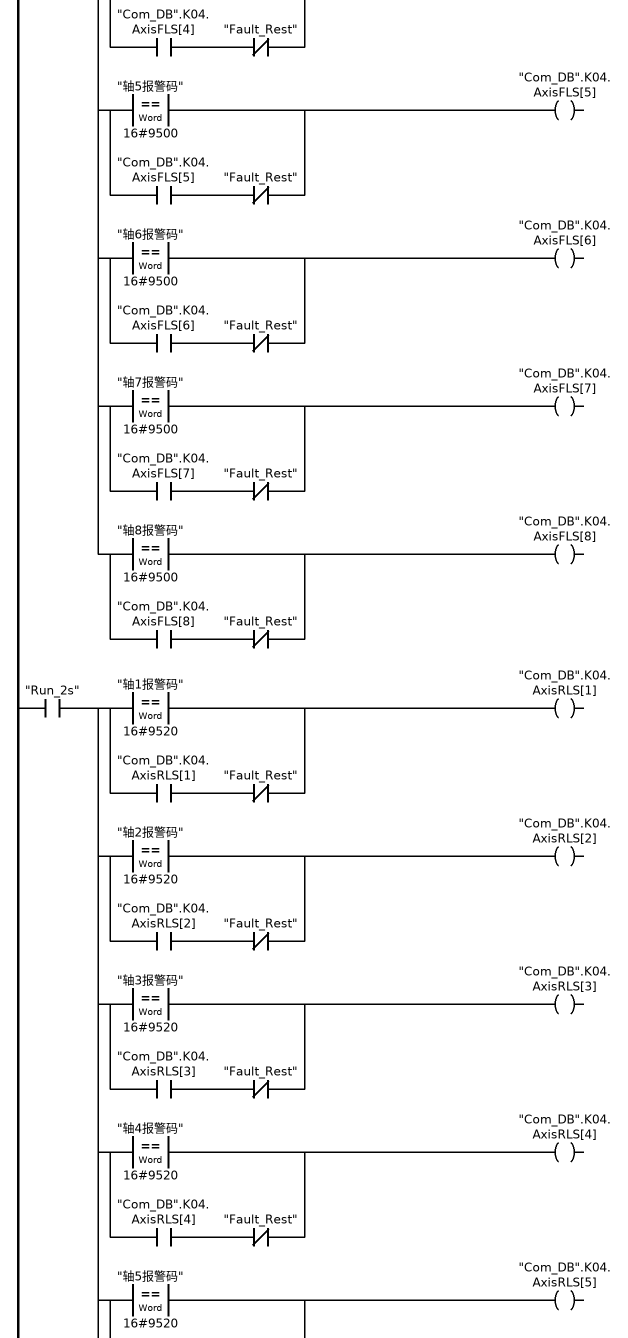
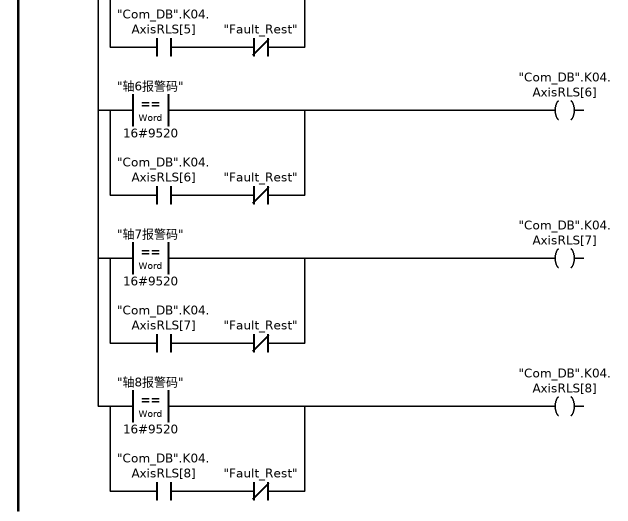
   "Com_DB".K04.AxisNoReady[1] := "Run_2s" AND ((NOT "轴1就绪" AND "轴1使能") OR ("Com_DB".K04.AxisNoReady[1] AND NOT "Fault_Rest"));
   "Com_DB".K04.AxisNoReady[2] := "Run_2s" AND ((NOT "轴2就绪" AND "轴2使能") OR ("Com_DB".K04.AxisNoReady[2] AND NOT "Fault_Rest"));
   "Com_DB".K04.AxisNoReady[3] := "Run_2s" AND ((NOT "轴3就绪" AND "轴3使能") OR ("Com_DB".K04.AxisNoReady[3] AND NOT "Fault_Rest"));
   "Com_DB".K04.AxisNoReady[4] := "Run_2s" AND ((NOT "轴4就绪" AND "轴4使能") OR ("Com_DB".K04.AxisNoReady[4] AND NOT "Fault_Rest"));
   "Com_DB".K04.AxisNoReady[5] := "Run_2s" AND ((NOT "轴5就绪" AND "轴5使能") OR ("Com_DB".K04.AxisNoReady[5] AND NOT "Fault_Rest"));
   "Com_DB".K04.AxisNoReady[6] := "Run_2s" AND ((NOT "轴6就绪" AND "轴6使能") OR ("Com_DB".K04.AxisNoReady[6] AND NOT "Fault_Rest"));
   "Com_DB".K04.AxisNoReady[7] := "Run_2s" AND ((NOT "轴7就绪" AND "轴7使能") OR ("Com_DB".K04.AxisNoReady[7] AND NOT "Fault_Rest"));
   "Com_DB".K04.AxisNoReady[8] := "Run_2s" AND ((NOT "轴8就绪" AND "轴8使能") OR ("Com_DB".K04.AxisNoReady[8] AND NOT "Fault_Rest"));
   #_w1 := "Run_2s" AND (("Com_DB".K07.Axis1Start AND NOT "轴1到达") OR ("Com_DB".K04.AxisNoRun[1] AND NOT "Fault_Rest"));
   "Com_DB".K04.AxisNoRun[1] := #_w1 AND "Com_DB".K04.AxisNoRunTon[1].Q;
   "Com_DB".K04.AxisNoRunTon[1].TON(IN := #_w1, PT := T#2S);   // TON coil
   #_w2 := "Run_2s" AND (("Com_DB".K07.Axis2Start AND NOT "轴2到达") OR ("Com_DB".K04.AxisNoRun[2] AND NOT "Fault_Rest"));
   "Com_DB".K04.AxisNoRun[2] := #_w2 AND "Com_DB".K04.AxisNoRunTon[2].Q;
   "Com_DB".K04.AxisNoRunTon[2].TON(IN := #_w2, PT := T#2S);   // TON coil
   #_w3 := "Run_2s" AND (("Com_DB".K07.Axis3Start AND NOT "轴3到达") OR ("Com_DB".K04.AxisNoRun[3] AND NOT "Fault_Rest"));
   "Com_DB".K04.AxisNoRun[3] := #_w3 AND "Com_DB".K04.AxisNoRunTon[3].Q;
   "Com_DB".K04.AxisNoRunTon[3].TON(IN := #_w3, PT := T#2S);   // TON coil
   #_w4 := "Run_2s" AND (("Com_DB".K07.Axis4Start AND NOT "轴4到达") OR ("Com_DB".K04.AxisNoRun[4] AND NOT "Fault_Rest"));
   "Com_DB".K04.AxisNoRun[4] := #_w4 AND "Com_DB".K04.AxisNoRunTon[4].Q;
   "Com_DB".K04.AxisNoRunTon[4].TON(IN := #_w4, PT := T#2S);   // TON coil
   #_w5 := "Run_2s" AND (("Com_DB".K07.Axis5Start AND NOT "轴5到达") OR ("Com_DB".K04.AxisNoRun[5] AND NOT "Fault_Rest"));
   "Com_DB".K04.AxisNoRun[5] := #_w5 AND "Com_DB".K04.AxisNoRunTon[5].Q;
   "Com_DB".K04.AxisNoRunTon[5].TON(IN := #_w5, PT := T#2S);   // TON coil
   #_w6 := "Run_2s" AND (("Com_DB".K07.Axis6Start AND NOT "轴6到达") OR ("Com_DB".K04.AxisNoRun[6] AND NOT "Fault_Rest"));
   "Com_DB".K04.AxisNoRun[6] := #_w6 AND "Com_DB".K04.AxisNoRunTon[6].Q;
   "Com_DB".K04.AxisNoRunTon[6].TON(IN := #_w6, PT := T#2S);   // TON coil
   #_w7 := "Run_2s" AND (("Com_DB".K07.Axis7Start AND NOT "轴7到达") OR ("Com_DB".K04.AxisNoRun[7] AND NOT "Fault_Rest"));
   "Com_DB".K04.AxisNoRun[7] := #_w7 AND "Com_DB".K04.AxisNoRunTon[7].Q;
   "Com_DB".K04.AxisNoRunTon[7].TON(IN := #_w7, PT := T#2S);   // TON coil
   #_w8 := "Run_2s" AND (("Com_DB".K07.Axis8Start AND NOT "轴8到达") OR ("Com_DB".K04.AxisNoRun[8] AND NOT "Fault_Rest"));
   "Com_DB".K04.AxisNoRun[8] := #_w8 AND "Com_DB".K04.AxisNoRunTon[8].Q;
   "Com_DB".K04.AxisNoRunTon[8].TON(IN := #_w8, PT := T#2S);   // TON coil
   "Com_DB".K04.AxisHomeALM[1] := "Run_2s" AND (NOT "轴1原点" OR ("Com_DB".K04.AxisHomeALM[1] AND NOT "Fault_Rest"));
   "Com_DB".K04.AxisHomeALM[2] := "Run_2s" AND (NOT "轴2原点" OR ("Com_DB".K04.AxisHomeALM[2] AND NOT "Fault_Rest"));
   "Com_DB".K04.AxisHomeALM[3] := "Run_2s" AND (NOT "轴3原点" OR ("Com_DB".K04.AxisHomeALM[3] AND NOT "Fault_Rest"));
   "Com_DB".K04.AxisHomeALM[4] := "Run_2s" AND (NOT "轴4原点" OR ("Com_DB".K04.AxisHomeALM[4] AND NOT "Fault_Rest"));
   "Com_DB".K04.AxisHomeALM[5] := "Run_2s" AND (NOT "轴5原点" OR ("Com_DB".K04.AxisHomeALM[5] AND NOT "Fault_Rest"));
   "Com_DB".K04.AxisHomeALM[6] := "Run_2s" AND (NOT "轴6原点" OR ("Com_DB".K04.AxisHomeALM[6] AND NOT "Fault_Rest"));
   "Com_DB".K04.AxisHomeALM[7] := "Run_2s" AND (NOT "轴7原点" OR ("Com_DB".K04.AxisHomeALM[7] AND NOT "Fault_Rest"));
   "Com_DB".K04.AxisHomeALM[8] := "Run_2s" AND (NOT "轴8原点" OR ("Com_DB".K04.AxisHomeALM[8] AND NOT "Fault_Rest"));
   "Com_DB".K04.AxisFLS[1] := "Run_2s" AND (("轴1报警码" = 16#9500) OR ("Com_DB".K04.AxisFLS[1] AND NOT "Fault_Rest"));
   "Com_DB".K04.AxisFLS[2] := "Run_2s" AND (("轴2报警码" = 16#9500) OR ("Com_DB".K04.AxisFLS[2] AND NOT "Fault_Rest"));
   "Com_DB".K04.AxisFLS[3] := "Run_2s" AND (("轴3报警码" = 16#9500) OR ("Com_DB".K04.AxisFLS[3] AND NOT "Fault_Rest"));
   "Com_DB".K04.AxisFLS[4] := "Run_2s" AND (("轴4报警码" = 16#9500) OR ("Com_DB".K04.AxisFLS[4] AND NOT "Fault_Rest"));
   "Com_DB".K04.AxisFLS[5] := "Run_2s" AND (("轴5报警码" = 16#9500) OR ("Com_DB".K04.AxisFLS[5] AND NOT "Fault_Rest"));
   "Com_DB".K04.AxisFLS[6] := "Run_2s" AND (("轴6报警码" = 16#9500) OR ("Com_DB".K04.AxisFLS[6] AND NOT "Fault_Rest"));
   "Com_DB".K04.AxisFLS[7] := "Run_2s" AND (("轴7报警码" = 16#9500) OR ("Com_DB".K04.AxisFLS[7] AND NOT "Fault_Rest"));
   "Com_DB".K04.AxisFLS[8] := "Run_2s" AND (("轴8报警码" = 16#9500) OR ("Com_DB".K04.AxisFLS[8] AND NOT "Fault_Rest"));
   "Com_DB".K04.AxisRLS[1] := "Run_2s" AND (("轴1报警码" = 16#9520) OR ("Com_DB".K04.AxisRLS[1] AND NOT "Fault_Rest"));
   "Com_DB".K04.AxisRLS[2] := "Run_2s" AND (("轴2报警码" = 16#9520) OR ("Com_DB".K04.AxisRLS[2] AND NOT "Fault_Rest"));
   "Com_DB".K04.AxisRLS[3] := "Run_2s" AND (("轴3报警码" = 16#9520) OR ("Com_DB".K04.AxisRLS[3] AND NOT "Fault_Rest"));
   "Com_DB".K04.AxisRLS[4] := "Run_2s" AND (("轴4报警码" = 16#9520) OR ("Com_DB".K04.AxisRLS[4] AND NOT "Fault_Rest"));
   "Com_DB".K04.AxisRLS[5] := "Run_2s" AND (("轴5报警码" = 16#9520) OR ("Com_DB".K04.AxisRLS[5] AND NOT "Fault_Rest"));
   "Com_DB".K04.AxisRLS[6] := "Run_2s" AND (("轴6报警码" = 16#9520) OR ("Com_DB".K04.AxisRLS[6] AND NOT "Fault_Rest"));
   "Com_DB".K04.AxisRLS[7] := "Run_2s" AND (("轴7报警码" = 16#9520) OR ("Com_DB".K04.AxisRLS[7] AND NOT "Fault_Rest"));
   "Com_DB".K04.AxisRLS[8] := "Run_2s" AND (("轴8报警码" = 16#9520) OR ("Com_DB".K04.AxisRLS[8] AND NOT "Fault_Rest"));
END_REGION

REGION Network 10: 机器人报警16个
END_REGION

REGION Network 11: 视觉报警16个
END_REGION

REGION Network 12: 通信报警16个
END_REGION

REGION Network 13: 模拟量故障16个
END_REGION

REGION Network 14: 其它报警32个
END_REGION

REGION Network 15: 传感器故障96个
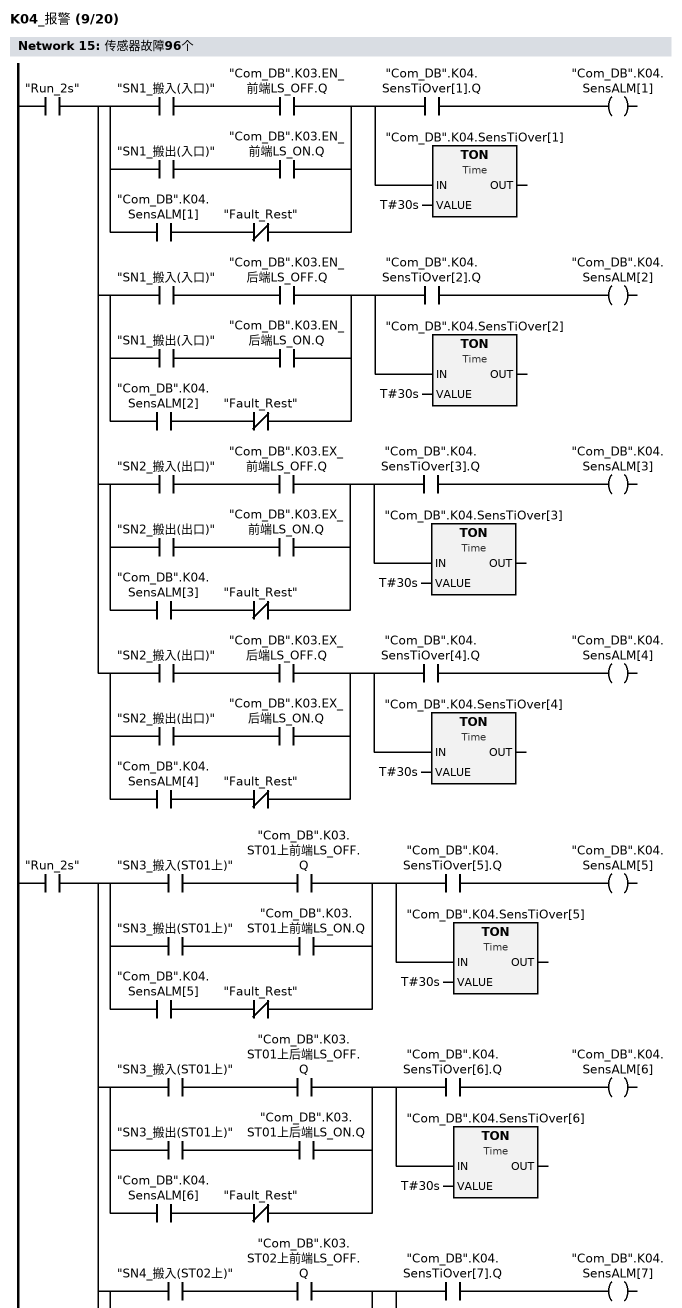
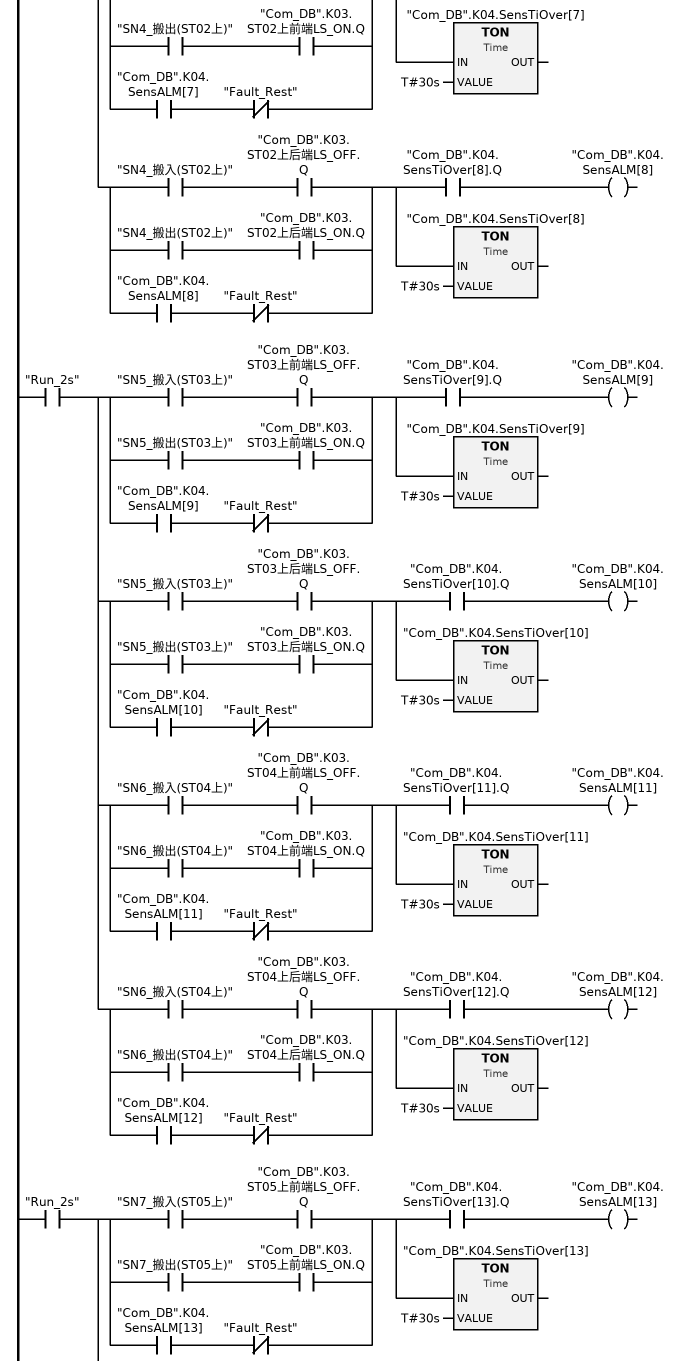
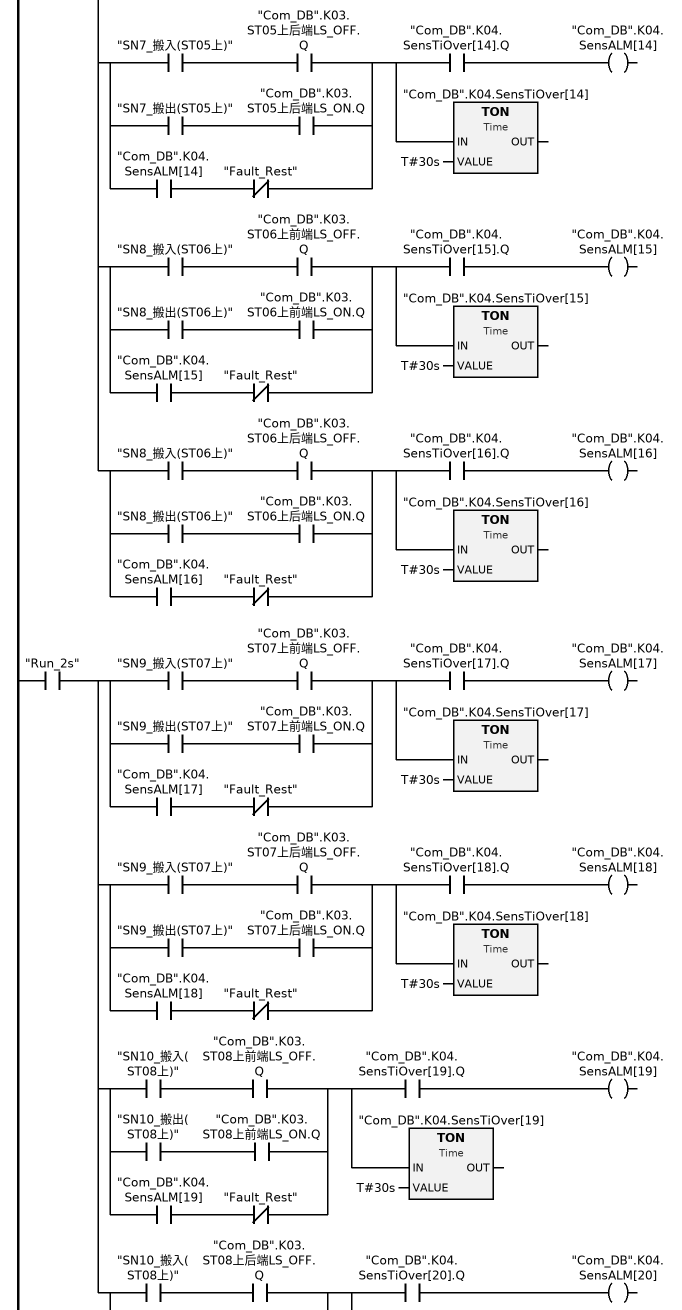
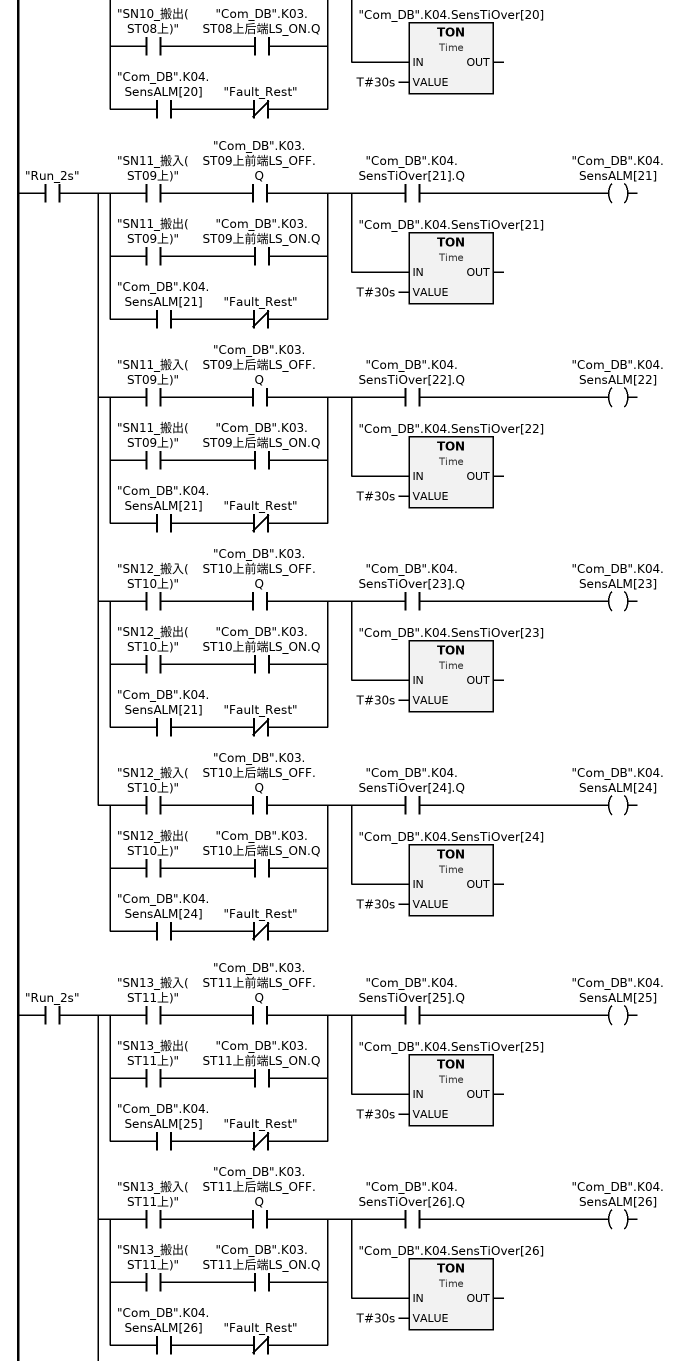
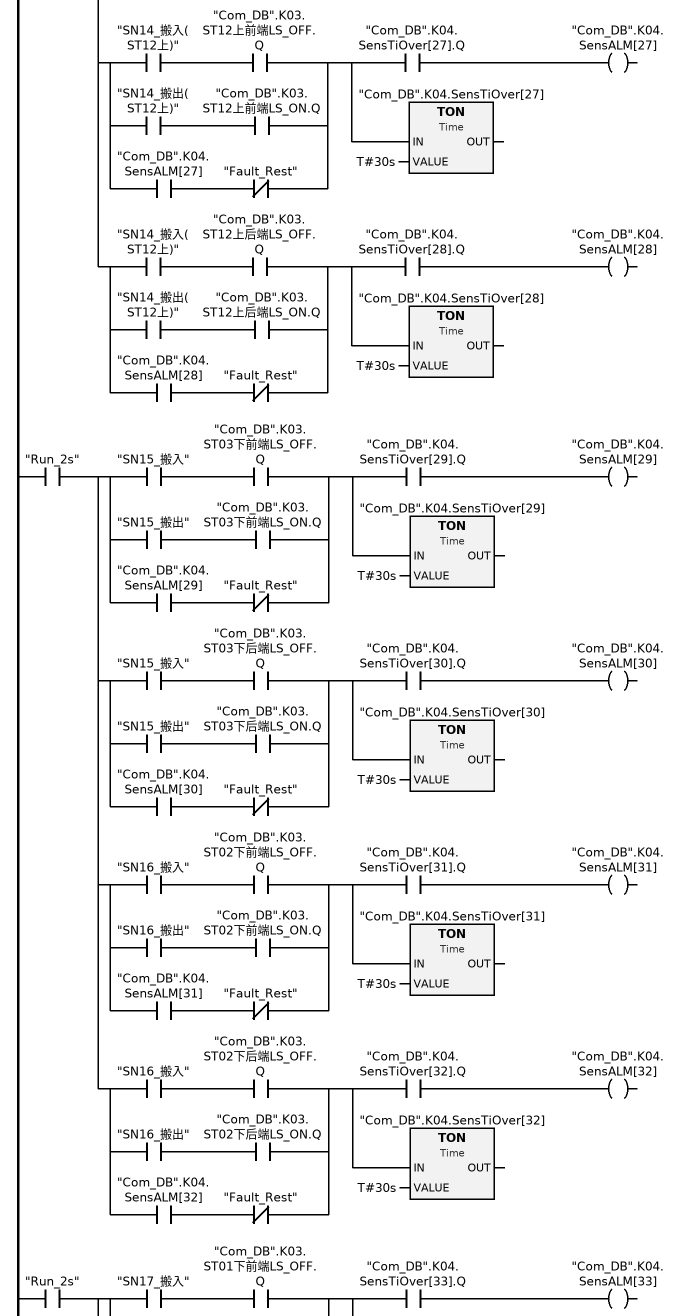
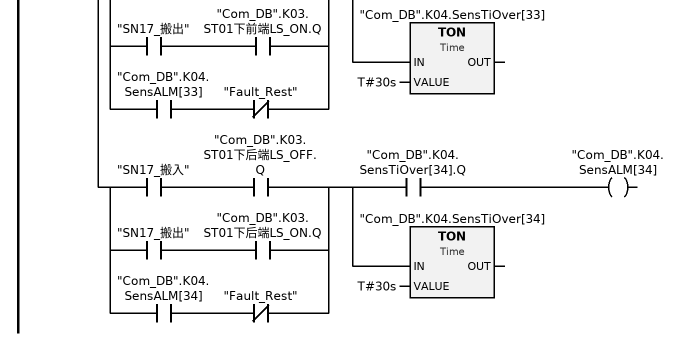
   #_w1 := "Run_2s" AND (("SN1_搬入(入口)" AND "Com_DB".K03.EN_前端LS_OFF.Q) OR ("SN1_搬出(入口)" AND "Com_DB".K03.EN_前端LS_ON.Q) OR ("Com_DB".K04.SensALM[1] AND NOT "Fault_Rest"));
   "Com_DB".K04.SensALM[1] := #_w1 AND "Com_DB".K04.SensTiOver[1].Q;
   "Com_DB".K04.SensTiOver[1].TON(IN := #_w1, PT := T#30s);   // TON coil
   #_w2 := "Run_2s" AND (("SN1_搬入(入口)" AND "Com_DB".K03.EN_后端LS_OFF.Q) OR ("SN1_搬出(入口)" AND "Com_DB".K03.EN_后端LS_ON.Q) OR ("Com_DB".K04.SensALM[2] AND NOT "Fault_Rest"));
   "Com_DB".K04.SensALM[2] := #_w2 AND "Com_DB".K04.SensTiOver[2].Q;
   "Com_DB".K04.SensTiOver[2].TON(IN := #_w2, PT := T#30s);   // TON coil
   #_w3 := "Run_2s" AND (("SN2_搬入(出口)" AND "Com_DB".K03.EX_前端LS_OFF.Q) OR ("SN2_搬出(出口)" AND "Com_DB".K03.EX_前端LS_ON.Q) OR ("Com_DB".K04.SensALM[3] AND NOT "Fault_Rest"));
   "Com_DB".K04.SensALM[3] := #_w3 AND "Com_DB".K04.SensTiOver[3].Q;
   "Com_DB".K04.SensTiOver[3].TON(IN := #_w3, PT := T#30s);   // TON coil
   #_w4 := "Run_2s" AND (("SN2_搬入(出口)" AND "Com_DB".K03.EX_后端LS_OFF.Q) OR ("SN2_搬出(出口)" AND "Com_DB".K03.EX_后端LS_ON.Q) OR ("Com_DB".K04.SensALM[4] AND NOT "Fault_Rest"));
   "Com_DB".K04.SensALM[4] := #_w4 AND "Com_DB".K04.SensTiOver[4].Q;
   "Com_DB".K04.SensTiOver[4].TON(IN := #_w4, PT := T#30s);   // TON coil
   #_w5 := "Run_2s" AND (("SN3_搬入(ST01上)" AND "Com_DB".K03.ST01上前端LS_OFF.Q) OR ("SN3_搬出(ST01上)" AND "Com_DB".K03.ST01上前端LS_ON.Q) OR ("Com_DB".K04.SensALM[5] AND NOT "Fault_Rest"));
   "Com_DB".K04.SensALM[5] := #_w5 AND "Com_DB".K04.SensTiOver[5].Q;
   "Com_DB".K04.SensTiOver[5].TON(IN := #_w5, PT := T#30s);   // TON coil
   #_w6 := "Run_2s" AND (("SN3_搬入(ST01上)" AND "Com_DB".K03.ST01上后端LS_OFF.Q) OR ("SN3_搬出(ST01上)" AND "Com_DB".K03.ST01上后端LS_ON.Q) OR ("Com_DB".K04.SensALM[6] AND NOT "Fault_Rest"));
   "Com_DB".K04.SensALM[6] := #_w6 AND "Com_DB".K04.SensTiOver[6].Q;
   "Com_DB".K04.SensTiOver[6].TON(IN := #_w6, PT := T#30s);   // TON coil
   #_w7 := "Run_2s" AND (("SN4_搬入(ST02上)" AND "Com_DB".K03.ST02上前端LS_OFF.Q) OR ("SN4_搬出(ST02上)" AND "Com_DB".K03.ST02上前端LS_ON.Q) OR ("Com_DB".K04.SensALM[7] AND NOT "Fault_Rest"));
   "Com_DB".K04.SensALM[7] := #_w7 AND "Com_DB".K04.SensTiOver[7].Q;
   "Com_DB".K04.SensTiOver[7].TON(IN := #_w7, PT := T#30s);   // TON coil
   #_w8 := "Run_2s" AND (("SN4_搬入(ST02上)" AND "Com_DB".K03.ST02上后端LS_OFF.Q) OR ("SN4_搬出(ST02上)" AND "Com_DB".K03.ST02上后端LS_ON.Q) OR ("Com_DB".K04.SensALM[8] AND NOT "Fault_Rest"));
   "Com_DB".K04.SensALM[8] := #_w8 AND "Com_DB".K04.SensTiOver[8].Q;
   "Com_DB".K04.SensTiOver[8].TON(IN := #_w8, PT := T#30s);   // TON coil
   #_w9 := "Run_2s" AND (("SN5_搬入(ST03上)" AND "Com_DB".K03.ST03上前端LS_OFF.Q) OR ("SN5_搬出(ST03上)" AND "Com_DB".K03.ST03上前端LS_ON.Q) OR ("Com_DB".K04.SensALM[9] AND NOT "Fault_Rest"));
   "Com_DB".K04.SensALM[9] := #_w9 AND "Com_DB".K04.SensTiOver[9].Q;
   "Com_DB".K04.SensTiOver[9].TON(IN := #_w9, PT := T#30s);   // TON coil
   #_w10 := "Run_2s" AND (("SN5_搬入(ST03上)" AND "Com_DB".K03.ST03上后端LS_OFF.Q) OR ("SN5_搬出(ST03上)" AND "Com_DB".K03.ST03上后端LS_ON.Q) OR ("Com_DB".K04.SensALM[10] AND NOT "Fault_Rest"));
   "Com_DB".K04.SensALM[10] := #_w10 AND "Com_DB".K04.SensTiOver[10].Q;
   "Com_DB".K04.SensTiOver[10].TON(IN := #_w10, PT := T#30s);   // TON coil
   #_w11 := "Run_2s" AND (("SN6_搬入(ST04上)" AND "Com_DB".K03.ST04上前端LS_OFF.Q) OR ("SN6_搬出(ST04上)" AND "Com_DB".K03.ST04上前端LS_ON.Q) OR ("Com_DB".K04.SensALM[11] AND NOT "Fault_Rest"));
   "Com_DB".K04.SensALM[11] := #_w11 AND "Com_DB".K04.SensTiOver[11].Q;
   "Com_DB".K04.SensTiOver[11].TON(IN := #_w11, PT := T#30s);   // TON coil
   #_w12 := "Run_2s" AND (("SN6_搬入(ST04上)" AND "Com_DB".K03.ST04上后端LS_OFF.Q) OR ("SN6_搬出(ST04上)" AND "Com_DB".K03.ST04上后端LS_ON.Q) OR ("Com_DB".K04.SensALM[12] AND NOT "Fault_Rest"));
   "Com_DB".K04.SensALM[12] := #_w12 AND "Com_DB".K04.SensTiOver[12].Q;
   "Com_DB".K04.SensTiOver[12].TON(IN := #_w12, PT := T#30s);   // TON coil
   #_w13 := "Run_2s" AND (("SN7_搬入(ST05上)" AND "Com_DB".K03.ST05上前端LS_OFF.Q) OR ("SN7_搬出(ST05上)" AND "Com_DB".K03.ST05上前端LS_ON.Q) OR ("Com_DB".K04.SensALM[13] AND NOT "Fault_Rest"));
   "Com_DB".K04.SensALM[13] := #_w13 AND "Com_DB".K04.SensTiOver[13].Q;
   "Com_DB".K04.SensTiOver[13].TON(IN := #_w13, PT := T#30s);   // TON coil
   #_w14 := "Run_2s" AND (("SN7_搬入(ST05上)" AND "Com_DB".K03.ST05上后端LS_OFF.Q) OR ("SN7_搬出(ST05上)" AND "Com_DB".K03.ST05上后端LS_ON.Q) OR ("Com_DB".K04.SensALM[14] AND NOT "Fault_Rest"));
   "Com_DB".K04.SensALM[14] := #_w14 AND "Com_DB".K04.SensTiOver[14].Q;
   "Com_DB".K04.SensTiOver[14].TON(IN := #_w14, PT := T#30s);   // TON coil
   #_w15 := "Run_2s" AND (("SN8_搬入(ST06上)" AND "Com_DB".K03.ST06上前端LS_OFF.Q) OR ("SN8_搬出(ST06上)" AND "Com_DB".K03.ST06上前端LS_ON.Q) OR ("Com_DB".K04.SensALM[15] AND NOT "Fault_Rest"));
   "Com_DB".K04.SensALM[15] := #_w15 AND "Com_DB".K04.SensTiOver[15].Q;
   "Com_DB".K04.SensTiOver[15].TON(IN := #_w15, PT := T#30s);   // TON coil
   #_w16 := "Run_2s" AND (("SN8_搬入(ST06上)" AND "Com_DB".K03.ST06上后端LS_OFF.Q) OR ("SN8_搬出(ST06上)" AND "Com_DB".K03.ST06上后端LS_ON.Q) OR ("Com_DB".K04.SensALM[16] AND NOT "Fault_Rest"));
   "Com_DB".K04.SensALM[16] := #_w16 AND "Com_DB".K04.SensTiOver[16].Q;
   "Com_DB".K04.SensTiOver[16].TON(IN := #_w16, PT := T#30s);   // TON coil
   #_w17 := "Run_2s" AND (("SN9_搬入(ST07上)" AND "Com_DB".K03.ST07上前端LS_OFF.Q) OR ("SN9_搬出(ST07上)" AND "Com_DB".K03.ST07上前端LS_ON.Q) OR ("Com_DB".K04.SensALM[17] AND NOT "Fault_Rest"));
   "Com_DB".K04.SensALM[17] := #_w17 AND "Com_DB".K04.SensTiOver[17].Q;
   "Com_DB".K04.SensTiOver[17].TON(IN := #_w17, PT := T#30s);   // TON coil
   #_w18 := "Run_2s" AND (("SN9_搬入(ST07上)" AND "Com_DB".K03.ST07上后端LS_OFF.Q) OR ("SN9_搬出(ST07上)" AND "Com_DB".K03.ST07上后端LS_ON.Q) OR ("Com_DB".K04.SensALM[18] AND NOT "Fault_Rest"));
   "Com_DB".K04.SensALM[18] := #_w18 AND "Com_DB".K04.SensTiOver[18].Q;
   "Com_DB".K04.SensTiOver[18].TON(IN := #_w18, PT := T#30s);   // TON coil
   #_w19 := "Run_2s" AND (("SN10_搬入(ST08上)" AND "Com_DB".K03.ST08上前端LS_OFF.Q) OR ("SN10_搬出(ST08上)" AND "Com_DB".K03.ST08上前端LS_ON.Q) OR ("Com_DB".K04.SensALM[19] AND NOT "Fault_Rest"));
   "Com_DB".K04.SensALM[19] := #_w19 AND "Com_DB".K04.SensTiOver[19].Q;
   "Com_DB".K04.SensTiOver[19].TON(IN := #_w19, PT := T#30s);   // TON coil
   #_w20 := "Run_2s" AND (("SN10_搬入(ST08上)" AND "Com_DB".K03.ST08上后端LS_OFF.Q) OR ("SN10_搬出(ST08上)" AND "Com_DB".K03.ST08上后端LS_ON.Q) OR ("Com_DB".K04.SensALM[20] AND NOT "Fault_Rest"));
   "Com_DB".K04.SensALM[20] := #_w20 AND "Com_DB".K04.SensTiOver[20].Q;
   "Com_DB".K04.SensTiOver[20].TON(IN := #_w20, PT := T#30s);   // TON coil
   #_w21 := "Run_2s" AND (("SN11_搬入(ST09上)" AND "Com_DB".K03.ST09上前端LS_OFF.Q) OR ("SN11_搬出(ST09上)" AND "Com_DB".K03.ST09上前端LS_ON.Q) OR ("Com_DB".K04.SensALM[21] AND NOT "Fault_Rest"));
   "Com_DB".K04.SensALM[21] := #_w21 AND "Com_DB".K04.SensTiOver[21].Q;
   "Com_DB".K04.SensTiOver[21].TON(IN := #_w21, PT := T#30s);   // TON coil
   #_w22 := "Run_2s" AND (("SN11_搬入(ST09上)" AND "Com_DB".K03.ST09上后端LS_OFF.Q) OR ("SN11_搬出(ST09上)" AND "Com_DB".K03.ST09上后端LS_ON.Q) OR ("Com_DB".K04.SensALM[21] AND NOT "Fault_Rest"));
   "Com_DB".K04.SensALM[22] := #_w22 AND "Com_DB".K04.SensTiOver[22].Q;
   "Com_DB".K04.SensTiOver[22].TON(IN := #_w22, PT := T#30s);   // TON coil
   #_w23 := "Run_2s" AND (("SN12_搬入(ST10上)" AND "Com_DB".K03.ST10上前端LS_OFF.Q) OR ("SN12_搬出(ST10上)" AND "Com_DB".K03.ST10上前端LS_ON.Q) OR ("Com_DB".K04.SensALM[21] AND NOT "Fault_Rest"));
   "Com_DB".K04.SensALM[23] := #_w23 AND "Com_DB".K04.SensTiOver[23].Q;
   "Com_DB".K04.SensTiOver[23].TON(IN := #_w23, PT := T#30s);   // TON coil
   #_w24 := "Run_2s" AND (("SN12_搬入(ST10上)" AND "Com_DB".K03.ST10上后端LS_OFF.Q) OR ("SN12_搬出(ST10上)" AND "Com_DB".K03.ST10上后端LS_ON.Q) OR ("Com_DB".K04.SensALM[24] AND NOT "Fault_Rest"));
   "Com_DB".K04.SensALM[24] := #_w24 AND "Com_DB".K04.SensTiOver[24].Q;
   "Com_DB".K04.SensTiOver[24].TON(IN := #_w24, PT := T#30s);   // TON coil
   #_w25 := "Run_2s" AND (("SN13_搬入(ST11上)" AND "Com_DB".K03.ST11上前端LS_OFF.Q) OR ("SN13_搬出(ST11上)" AND "Com_DB".K03.ST11上前端LS_ON.Q) OR ("Com_DB".K04.SensALM[25] AND NOT "Fault_Rest"));
   "Com_DB".K04.SensALM[25] := #_w25 AND "Com_DB".K04.SensTiOver[25].Q;
   "Com_DB".K04.SensTiOver[25].TON(IN := #_w25, PT := T#30s);   // TON coil
   #_w26 := "Run_2s" AND (("SN13_搬入(ST11上)" AND "Com_DB".K03.ST11上后端LS_OFF.Q) OR ("SN13_搬出(ST11上)" AND "Com_DB".K03.ST11上后端LS_ON.Q) OR ("Com_DB".K04.SensALM[26] AND NOT "Fault_Rest"));
   "Com_DB".K04.SensALM[26] := #_w26 AND "Com_DB".K04.SensTiOver[26].Q;
   "Com_DB".K04.SensTiOver[26].TON(IN := #_w26, PT := T#30s);   // TON coil
   #_w27 := "Run_2s" AND (("SN14_搬入(ST12上)" AND "Com_DB".K03.ST12上前端LS_OFF.Q) OR ("SN14_搬出(ST12上)" AND "Com_DB".K03.ST12上前端LS_ON.Q) OR ("Com_DB".K04.SensALM[27] AND NOT "Fault_Rest"));
   "Com_DB".K04.SensALM[27] := #_w27 AND "Com_DB".K04.SensTiOver[27].Q;
   "Com_DB".K04.SensTiOver[27].TON(IN := #_w27, PT := T#30s);   // TON coil
   #_w28 := "Run_2s" AND (("SN14_搬入(ST12上)" AND "Com_DB".K03.ST12上后端LS_OFF.Q) OR ("SN14_搬出(ST12上)" AND "Com_DB".K03.ST12上后端LS_ON.Q) OR ("Com_DB".K04.SensALM[28] AND NOT "Fault_Rest"));
   "Com_DB".K04.SensALM[28] := #_w28 AND "Com_DB".K04.SensTiOver[28].Q;
   "Com_DB".K04.SensTiOver[28].TON(IN := #_w28, PT := T#30s);   // TON coil
   #_w29 := "Run_2s" AND (("SN15_搬入" AND "Com_DB".K03.ST03下前端LS_OFF.Q) OR ("SN15_搬出" AND "Com_DB".K03.ST03下前端LS_ON.Q) OR ("Com_DB".K04.SensALM[29] AND NOT "Fault_Rest"));
   "Com_DB".K04.SensALM[29] := #_w29 AND "Com_DB".K04.SensTiOver[29].Q;
   "Com_DB".K04.SensTiOver[29].TON(IN := #_w29, PT := T#30s);   // TON coil
   #_w30 := "Run_2s" AND (("SN15_搬入" AND "Com_DB".K03.ST03下后端LS_OFF.Q) OR ("SN15_搬出" AND "Com_DB".K03.ST03下后端LS_ON.Q) OR ("Com_DB".K04.SensALM[30] AND NOT "Fault_Rest"));
   "Com_DB".K04.SensALM[30] := #_w30 AND "Com_DB".K04.SensTiOver[30].Q;
   "Com_DB".K04.SensTiOver[30].TON(IN := #_w30, PT := T#30s);   // TON coil
   #_w31 := "Run_2s" AND (("SN16_搬入" AND "Com_DB".K03.ST02下前端LS_OFF.Q) OR ("SN16_搬出" AND "Com_DB".K03.ST02下前端LS_ON.Q) OR ("Com_DB".K04.SensALM[31] AND NOT "Fault_Rest"));
   "Com_DB".K04.SensALM[31] := #_w31 AND "Com_DB".K04.SensTiOver[31].Q;
   "Com_DB".K04.SensTiOver[31].TON(IN := #_w31, PT := T#30s);   // TON coil
   #_w32 := "Run_2s" AND (("SN16_搬入" AND "Com_DB".K03.ST02下后端LS_OFF.Q) OR ("SN16_搬出" AND "Com_DB".K03.ST02下后端LS_ON.Q) OR ("Com_DB".K04.SensALM[32] AND NOT "Fault_Rest"));
   "Com_DB".K04.SensALM[32] := #_w32 AND "Com_DB".K04.SensTiOver[32].Q;
   "Com_DB".K04.SensTiOver[32].TON(IN := #_w32, PT := T#30s);   // TON coil
   #_w33 := "Run_2s" AND (("SN17_搬入" AND "Com_DB".K03.ST01下前端LS_OFF.Q) OR ("SN17_搬出" AND "Com_DB".K03.ST01下前端LS_ON.Q) OR ("Com_DB".K04.SensALM[33] AND NOT "Fault_Rest"));
   "Com_DB".K04.SensALM[33] := #_w33 AND "Com_DB".K04.SensTiOver[33].Q;
   "Com_DB".K04.SensTiOver[33].TON(IN := #_w33, PT := T#30s);   // TON coil
   #_w34 := "Run_2s" AND (("SN17_搬入" AND "Com_DB".K03.ST01下后端LS_OFF.Q) OR ("SN17_搬出" AND "Com_DB".K03.ST01下后端LS_ON.Q) OR ("Com_DB".K04.SensALM[34] AND NOT "Fault_Rest"));
   "Com_DB".K04.SensALM[34] := #_w34 AND "Com_DB".K04.SensTiOver[34].Q;
   "Com_DB".K04.SensTiOver[34].TON(IN := #_w34, PT := T#30s);   // TON coil
END_REGION

REGION Network 16: 动作异常48个
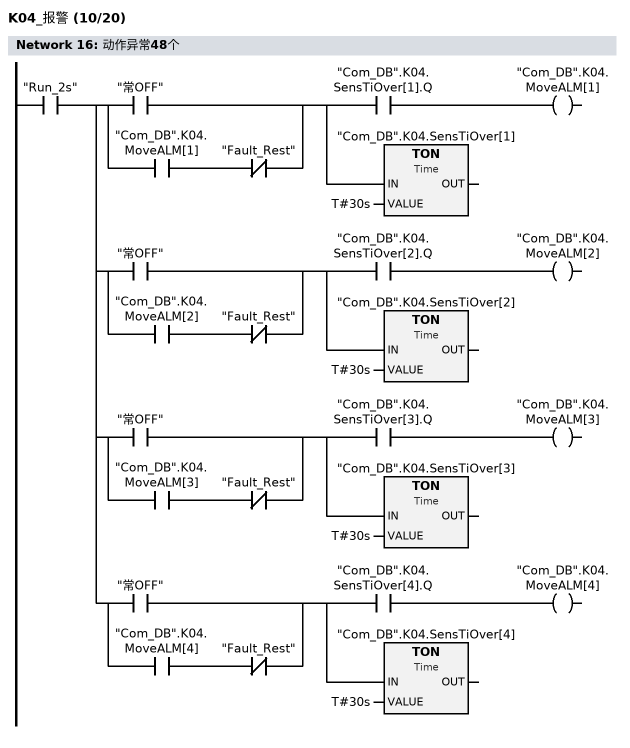
   #_w1 := "Run_2s" AND ("常OFF" OR ("Com_DB".K04.MoveALM[1] AND NOT "Fault_Rest"));
   "Com_DB".K04.MoveALM[1] := #_w1 AND "Com_DB".K04.SensTiOver[1].Q;
   "Com_DB".K04.SensTiOver[1].TON(IN := #_w1, PT := T#30s);   // TON coil
   #_w2 := "Run_2s" AND ("常OFF" OR ("Com_DB".K04.MoveALM[2] AND NOT "Fault_Rest"));
   "Com_DB".K04.MoveALM[2] := #_w2 AND "Com_DB".K04.SensTiOver[2].Q;
   "Com_DB".K04.SensTiOver[2].TON(IN := #_w2, PT := T#30s);   // TON coil
   #_w3 := "Run_2s" AND ("常OFF" OR ("Com_DB".K04.MoveALM[3] AND NOT "Fault_Rest"));
   "Com_DB".K04.MoveALM[3] := #_w3 AND "Com_DB".K04.SensTiOver[3].Q;
   "Com_DB".K04.SensTiOver[3].TON(IN := #_w3, PT := T#30s);   // TON coil
   #_w4 := "Run_2s" AND ("常OFF" OR ("Com_DB".K04.MoveALM[4] AND NOT "Fault_Rest"));
   "Com_DB".K04.MoveALM[4] := #_w4 AND "Com_DB".K04.SensTiOver[4].Q;
   "Com_DB".K04.SensTiOver[4].TON(IN := #_w4, PT := T#30s);   // TON coil
END_REGION

REGION Network 17: 报警数组汇总
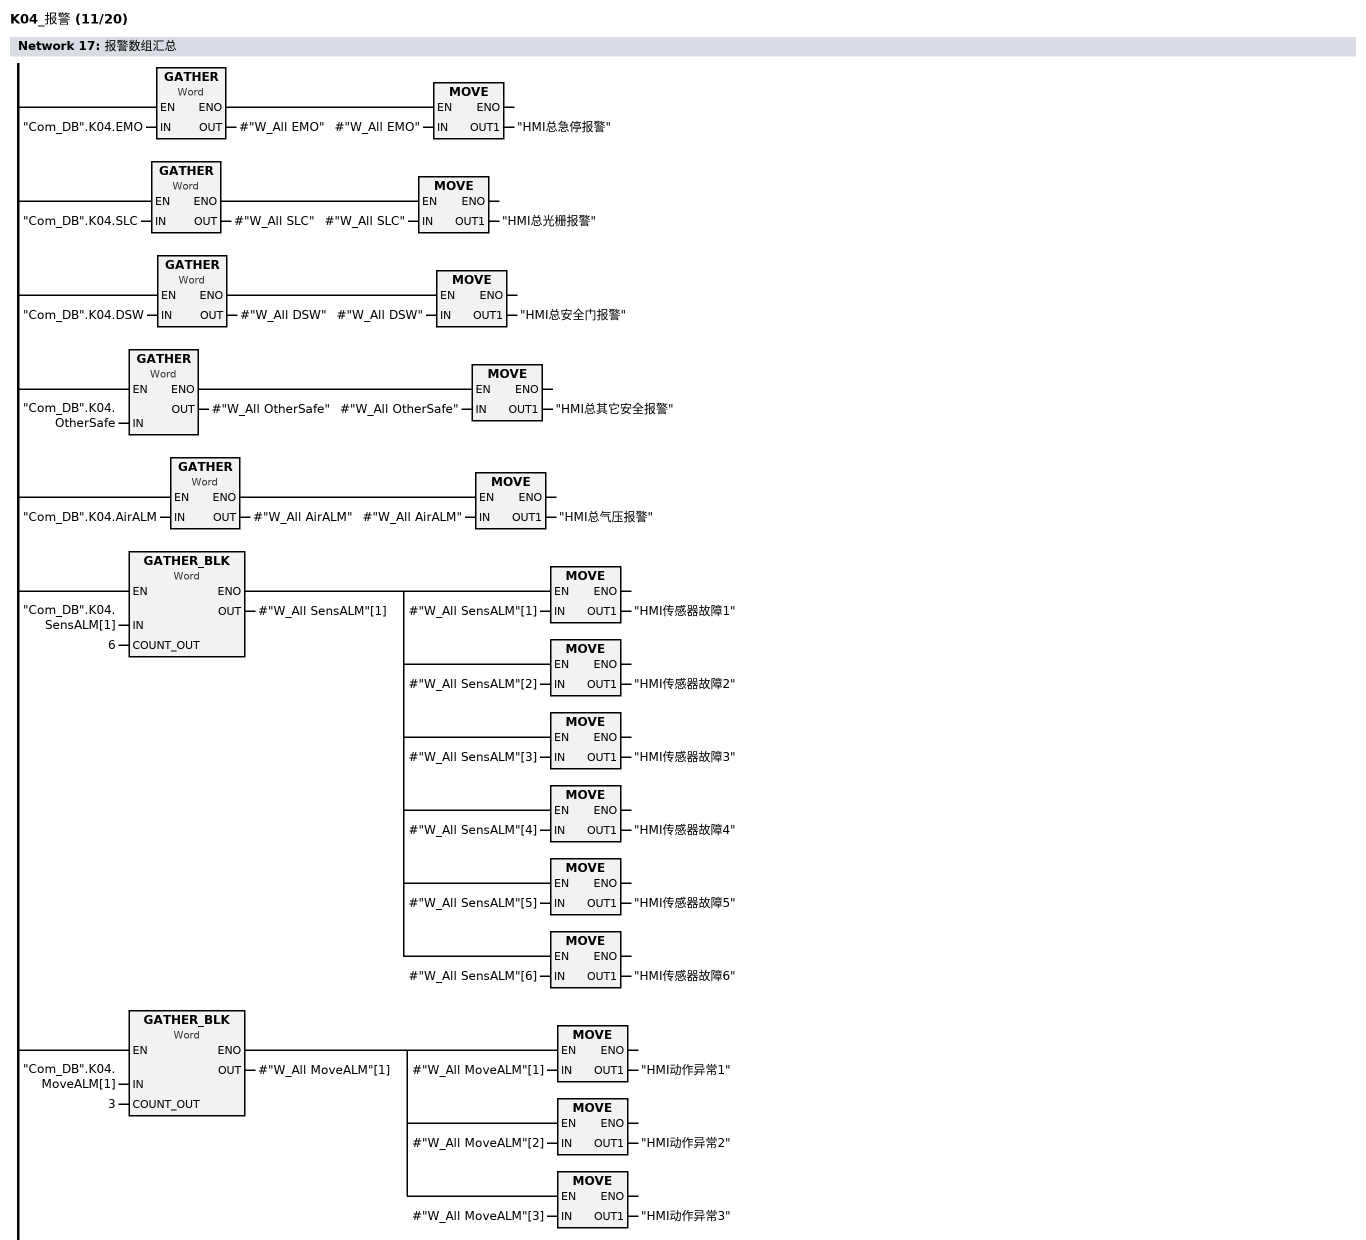
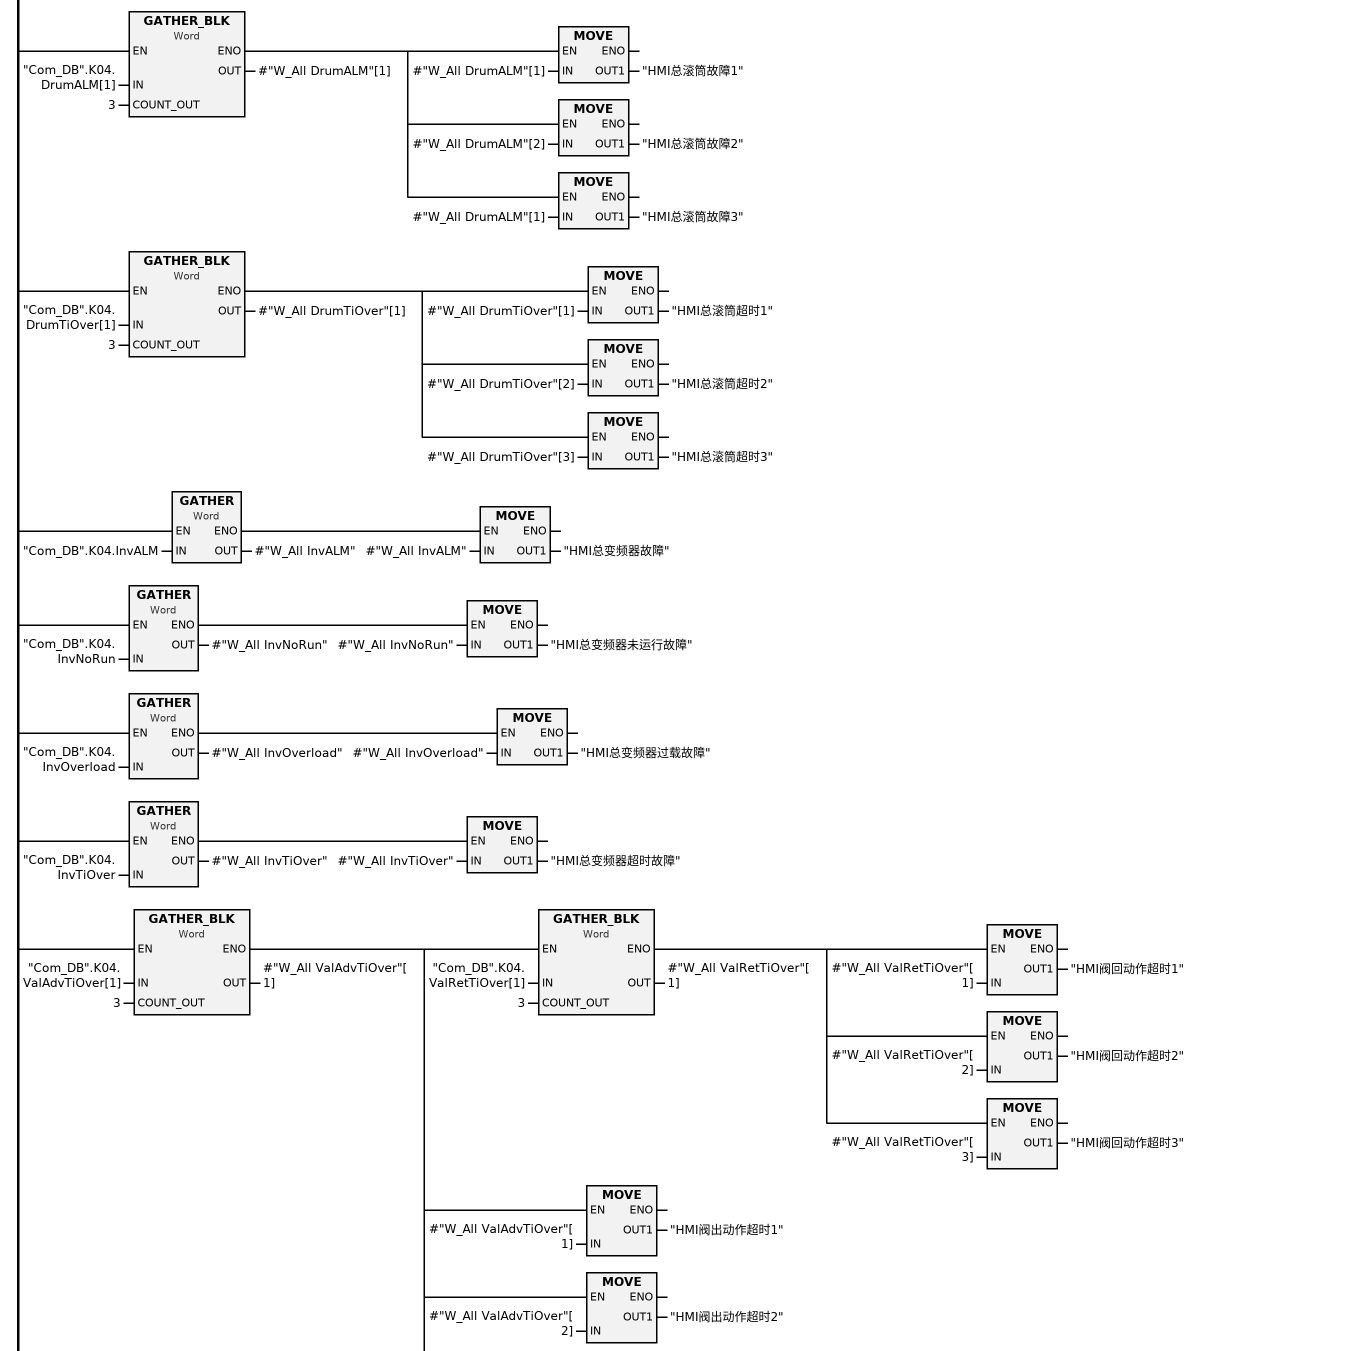
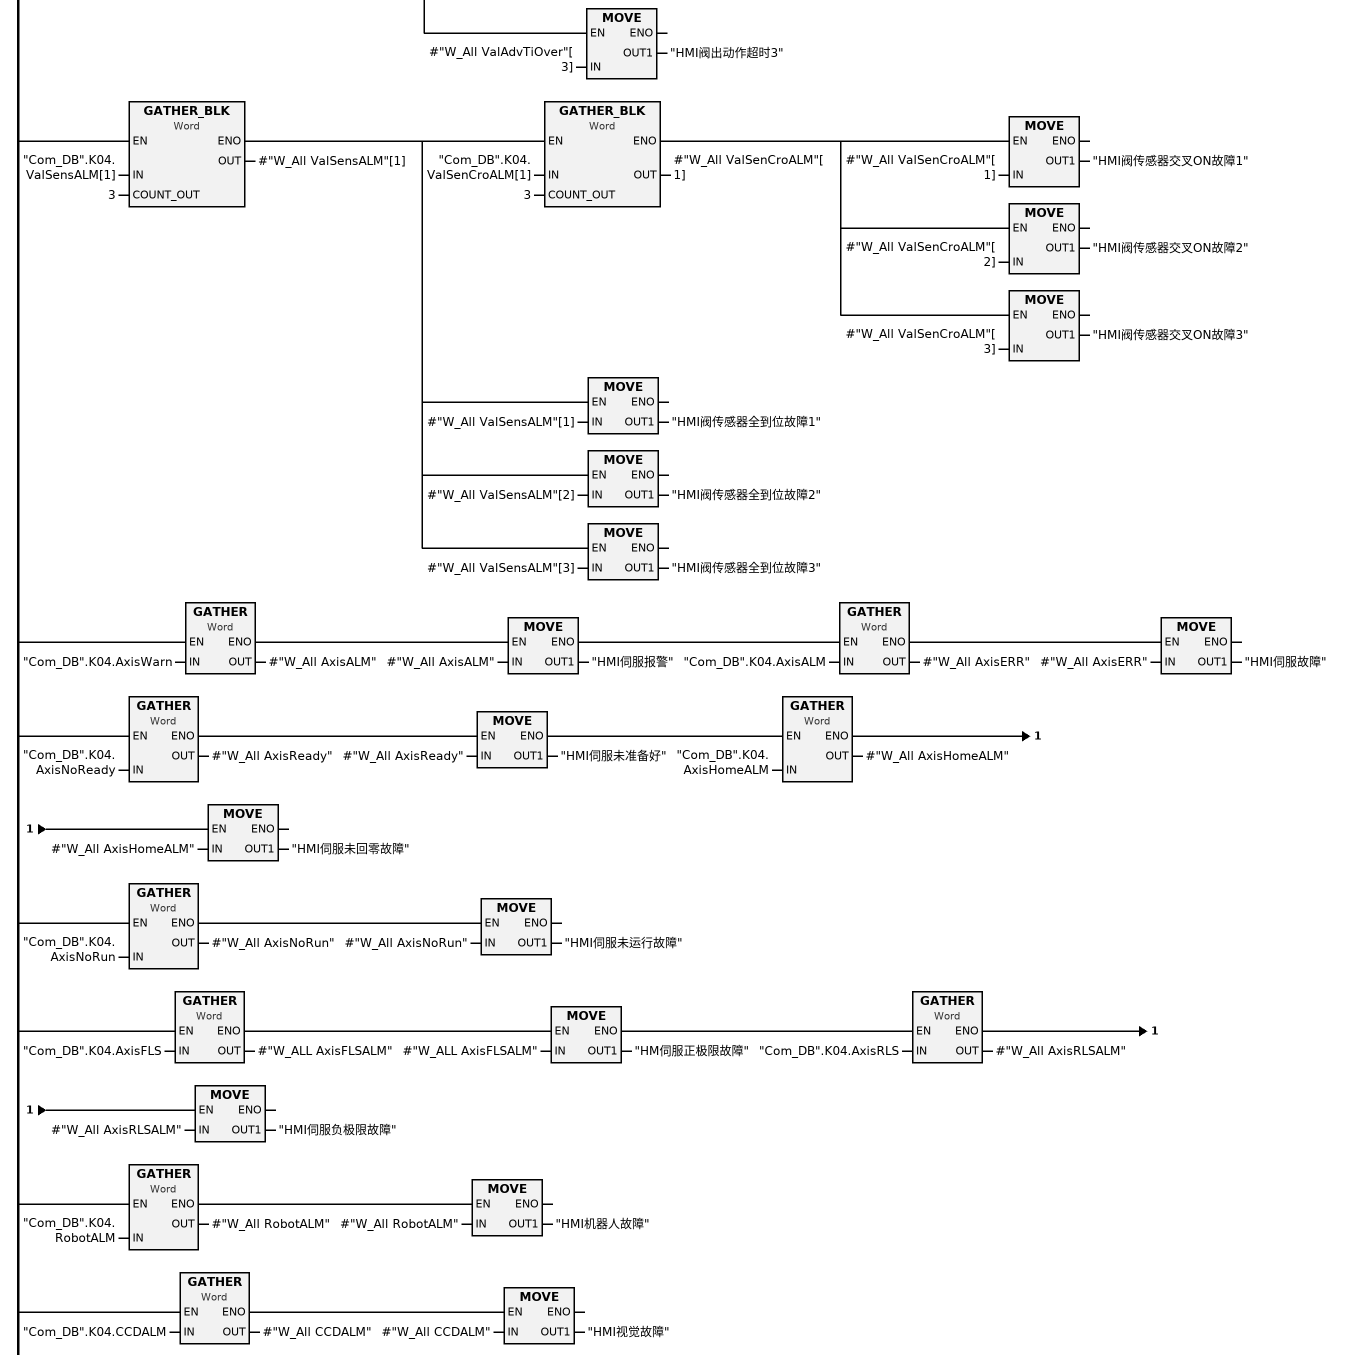
